Omron CX-Programmer project NewProject (CX-Programmer 9.76)

# PLC LQK19011ICM: CP1H XA
I/O table (CPU CP1H-XA40DR-A): rack 0 slot 0 CJ1W-SCU21

## Global symbols (name address type ; comment)
AI_SAW_CURRENT 200 CHANNEL  ; ANALOG.INPUT1.SAW.CURRENT
AI_TRANS_AXIS_DRIVE_VEL_FDBK 201 CHANNEL  ; AI.TRANSVERSE.AXIS.DRIVE.VELOCITY.FEEDBACK
AO_TRANS_VEL_REF 210 CHANNEL  ; TRANSVERSE.AXIS.VELOCITY.ANALOG.REFERENCE
0.05 BOOL  ; SPARE - Possible Zone Interference Limit Switch Input.
101 CHANNEL  ; @+ D205 &4 D205
1.03 BOOL  ; Spare
200 CHANNEL  ; Saw Motor Current Input
210 CHANNEL  ; Cross Travel Speed Refernce Command
40 CHANNEL  ; OI.SCALING.SAW.CURRENT.PART1
8.00 BOOL  ; Place holder for Automatic PID control request
A434.04 BOOL  ; Analog IO Initialised
D10009 CHANNEL  ; Spare
D1001 CHANNEL  ; Block 1 Data - Number of Blocks
D11040 CHANNEL  ; Operation Program Check Block 1 Slab 5 ID
D11050 CHANNEL  ; Operation Program Check Slab 6 ID
D11060 CHANNEL  ; Operation Program Check Slab ID
D11070 CHANNEL  ; Operation Program Check Slab 8 ID
D11080 CHANNEL  ; Operation Program Check Slab 9 ID
D11090 CHANNEL  ; Operation Program Check Slab 10 ID
D11100 CHANNEL  ; Operation Block 3 Slab 1 ID
D11110 CHANNEL  ; Operation Program Check Block 3 Slab 2 ID
D11120 CHANNEL  ; Operation Block 3 Slab 3 ID
D12301 CHANNEL  ; Operation Slab 31 Quantity
D12302 CHANNEL  ; Operation Program Check Block 7 Slab 31 Width
D200 CHANNEL  ; Number of Blocks Stored
D2002 CHANNEL  ; OPERATION.PROGRAM.CHECK.BLOCK1.SLAB2.SIZE
D201 CHANNEL  ; Operation Number of Words to Xfer
D202 CHANNEL  ; Captured Bumber of Blocks
D203 CHANNEL  ; Number of Blocks Difference
D204 CHANNEL  ; Slab Count Offset
D205 CHANNEL  ; Slab Word Count to Transfer
D3000 CHANNEL  ; Input Data Table Control Word
D3001 CHANNEL  ; Maximum Anaolg Input Value (Xm)
D3002 CHANNEL  ; Y0
D3003 CHANNEL  ; X1
D3004 CHANNEL  ; Maximum Output value
D3100 CHANNEL  ; Output Data Control Word
D3101 CHANNEL  ; Xm
D3102 CHANNEL  ; Y0
D3103 CHANNEL  ; X1
D3104 CHANNEL  ; Y1
D3106 CHANNEL  ; Interin feed rate calc word
D32 CHANNEL  ; OPERATION.AUTO.CYCLE.BLOCK.FIRST.CUT.WORKING.REAL
D3200 CHANNEL  ; Setpoint Input Data Table Control Word
D3201 CHANNEL  ; Maximum Input Setpoint
D3202 CHANNEL  ; Y0
D3203 CHANNEL  ; X1
D3204 CHANNEL  ; Y1
D34 CHANNEL  ; OP.CONTROL.VERTICAL.TARGET.SCALED
D3520 CHANNEL  ; PID Setpoint Scaled for PID
D3521 CHANNEL  ; PID Instruction Proportional Component
D3522 CHANNEL  ; PID Instruction Integral Component
D3523 CHANNEL  ; PID Instruction Derivative Component
D3524 CHANNEL  ; PID Instruction Period
D3525 CHANNEL  ; PID Instruction Control Word
D3526 CHANNEL  ; PID Instruction Input and Output Range Setting
D3527 CHANNEL  ; PID Instruction Output Minimum
D3528 CHANNEL  ; PID Instruction Output Maximum
D36 CHANNEL  ; OPERATION.AUTO.CYCLE.VERTICAL.HIGH/LOW/SPEED.SELECT
D40 CHANNEL  ; OP.CONTROL.CURRENT.BLOCK.HEIGHT.REAL
D400 CHANNEL  ; Working Floating Point First Cut Value Current Block
D4000 CHANNEL  ; OPERATION.AUTO.CYCLE.BLK.PTR
D4002 CHANNEL  ; OPERATION.AUTO.CYCLE.BLOCK.DATA.POINTER
D4004 CHANNEL  ; OPERATION.CURRENT.PROGRAM.SLAB.DATA.POINTER
D4006 CHANNEL  ; OPERATION.AUTO.CYCLE.SPARE
D4008 CHANNEL  ; OPERATION.AUTO.CYCLE.SPARE
D4010 CHANNEL  ; OPERATION.SLAB.POINTER.THIS.BLOCK
D4012 CHANNEL  ; OPERATION.AUTO.CYCLE.CURRENT.SLAB.CUT.COUNTER
D4014 CHANNEL  ; OPERATION.AUTO.CYCLE.SLAB.POINTER
D42 CHANNEL  ; OP.CONTROL.CURRENT.BLOCK.LENGTH
D44 CHANNEL  ; OP.CONTROL.AUTO.CYCLE.VERTICAL.TARGET
D46 CHANNEL  ; OP.CONTROL.AUTO.TRANSVERSE.TARGET.FORWARD
D48 CHANNEL  ; OP.CONTROL.TRANSVERSE.POSITION.TARGET.REAL
D480 CHANNEL  ; Ctl.PID.Output.Value
D484 CHANNEL  ; Saw Current Scaled for PID instruction use
D50 CHANNEL  ; OPERATION.AUTO.CYCLE.BLOCK.HEIGHT.REAL
D500 CHANNEL  ; First Cut Position Stored Float
D502 CHANNEL  ; Stored Slab Size Inches Float
D504 CHANNEL  ; Total Slab Size Float
D506 CHANNEL  ; Stored Kerf Size Total
D508 CHANNEL  ; Slab Total Size Calc'd
D510 CHANNEL  ; Total of First Cut Position and Slab Size
D512 CHANNEL  ; Final Calculated Position at Cut Finish of this Slab and this Block
D5120 CHANNEL  ; OI Long Axis Target
D52 CHANNEL  ; OPERATION.AUTO.CYCLE.BLOCK.TRANSVERSE.AXIS.FORWARD.STOP.POSITION
D5200 CHANNEL  ; Operation Long Axis Target Minimum
D54 CHANNEL  ; OPERATION.AUTO.CYCLE.BLOCK.FIRST.CUT.REAL
D5400 CHANNEL  ; OPERATION.LONG.TRAVEL.TARGET.WINDOW.PLUS
D5402 CHANNEL  ; OPERATION.LONG.TRAVEL.TARGET.WINDOW.MINUS
D5404 CHANNEL  ; OPERATION.LONG.TRAVEL.TARGET.WINDOW.SLABCUT.PLUS
D5406 CHANNEL  ; OPERATION.LONG.TRAVEL.TARGET.SLABCUT.MINUS
D5500 CHANNEL  ; OPERATION.AUTO.CYCLE.BLOCK.FIRST.CUT.REAL.SCALED
D5502 CHANNEL  ; OPERATION.AUTO.CYCLE.LON.INDEX.LOCATION.REAL.SCALED
D56 CHANNEL  ; OPERATION.AUTO.CYCLE.LONG.TARGET.KERF
D5600 CHANNEL  ; MC.TRANSVERSE.AXIS.POSITION.FEEDBACK.GB.SCALED.REAL
D58 CHANNEL  ; OPERATION.AUTO.CYCLE.ADD.KERF.TO.LOCATION.REAL
D6 CHANNEL  ; OPERATION.TRANSVERSE.AXIS.JOG.VELOCITY.REFERNCE.WORD
D60 CHANNEL  ; OPERATION.AUTO.CYCLE.LONG.INDEX.LOCATION.REAL
D6000 CHANNEL  ; MC.TRANSVERSE.AXIS.POSITION.FEEDBACK.RAW.REAL
D6002 CHANNEL  ; MC.TRANSVERSE.AXIS.POSITION.FEEDBACK.GB.SCALED.REAL
D6004 CHANNEL  ; MC.TRANSVERSE.AXIS.POSITION.PINION.REVOLUTIONS.REAL
D6006 CHANNEL  ; PI.EQUATION.PART.ONE
D6008 CHANNEL  ; PI.EQUATION.PART.TWO
D6012 CHANNEL  ; PI
D6014 CHANNEL  ; MC.TRANSVERSE.AXIS.PINION.CIRCUMFERENCE.INCHES.REAL
D66 CHANNEL  ; OPERATION.AUTO.CYCLE.CURRENT.SLAB.SIZE.REAL.RAW
D76 CHANNEL  ; OP.TRANSVERSE.AXIS.FORWARD.TARGET
D80 CHANNEL  ; Blade Kerf Raw Converted
D82 CHANNEL  ; Cut Depth Raw Converted
D84 CHANNEL  ; Cut Target Current Raw Converted
D86 CHANNEL  ; Current Slab Size Raw Converted
D97 CHANNEL  ; OP.CONTROL.AUTO.CYCLE.CURRENT.FIRST.CUT.LOCATION.LONG
D990 CHANNEL  ; PID Setpoint
H0.05 BOOL  ; OPERATION.ALARM.STATE.VALID
H0.11 BOOL  ; OPERATION.ALARM.RESET.COMMAND
H10.13 BOOL  ; MC.LONG.AXIS.STATE.VALID
H11.03 BOOL  ; VERTICAL.AXIS.DRIVE.NOT.OKAY
H11.07 BOOL  ; MC.VERTICAL.AXIS.JOG.PLUS
H11.08 BOOL  ; MC.VERTICAL.AXIS.JOG.MINUS
H11.13 BOOL  ; MC.VERTICAL.AXIS.DRIVE.RESET.ENABLED
H12.07 BOOL  ; MC.TRANSVERSE.AXIS.JOG.PLUS.INT
H12.08 BOOL  ; MC.TRANSVERSE.AXIS.JOG.NEG
H12.13 BOOL  ; MC.TRANSVERSE.AXIS.DRIVE.RESET.ENABLED
H13.04 BOOL  ; SAW.AUTO.RUN.UP.TIMER.DONE
H13.05 BOOL  ; OPERATION.AUTO.CYCLE.SAW.OVERCURRENT.ALARM
H13.06 BOOL  ; OPERATION.SAW.CURRENT.SENSING.CHECK.FAULT
H13.07 BOOL  ; OPERATION.SAW.MACHINE.STOP.COMMAND.ACTIVE
H13.08 BOOL  ; OPERATION.SAW.MACHINE.STOP.COMMAND.NOT ACTIVE
H13.13 BOOL  ; OPERATION.SAW.STATE.VALID
H13.15 BOOL  ; OP.ALARM.SAW.SOFT.START.FAULTED
H14.02 BOOL  ; WATER.FLOW.SHOULD.BE.ON
H14.03 BOOL  ; WATER.FLOW.IS.ON.AND.SHOULDN'T
H14.07 BOOL  ; OP.WATER.MACHINE.STOP.COMMAND.ACTIVE
H14.08 BOOL  ; OP.WATER.MACHINE.sTOP.COMMAND.NOT.ACTIVE
H14.13 BOOL  ; OPERATION.WATER.STATE.VALID
H14.14 BOOL  ; OP.ALARM.WATER.FLOW.ERROR
H16.13 BOOL  ; OPERATION.RECIPE.STATE.VALID
H16.14 BOOL  ; RECIPE.ERROR
H17.00 BOOL  ; Operation Auto Cycle State Invalid Over Time Alarm
H1.00 BOOL  ; OP.MODE.INDICATOR.ENABLED
H1.01 BOOL  ; OP.MODE.AUTO.PGM.CHECK.ACT
H1.02 BOOL  ; OP.MODE.AUTO.PGM.CHECK.CMP
H1.03 BOOL  ; LAST.BLOCK.CHECK
H1.14 BOOL  ; ALARM.RESEST.TRAP
H1.15 BOOL  ; MODE.AUTO.GATE.ALARM.TRIGGER
H2 CHANNEL  ; Cycle Start Bits
H20.04 BOOL  ; OPERATION.AUTO.CYCLE.LONG.AXIS.MOTION.READY
H20.05 BOOL  ; OPERATION.AUTO.CYCLE.LONG.AXIS.MOTION.ENABLED
H20.06 BOOL  ; OP.CONTROL.AUTO.CYCLE.INDEX.LONG.AXIS.COMMAND
H20.07 BOOL  ; OPERATION.AUTO.CYCLE.LONG.AXIS.INDEX.COMMAND.ACTIVE
H20.08 BOOL  ; OPERATION.LONG.AXIS.IN.POSITION.WINDOW.TOLERANCE
H20.09 BOOL  ; OPERATION.AUTO.CYCLE.LONG.AXIS.INDEX.COMMAND.COMPLETE
H20.10 BOOL  ; OPERATION.AUTO.CYCLE.LONG.AXIS.MOTION.SAFE
H20.11 BOOL  ; OPERATION.AUTO.CYCLE.LONG.AXIS.MOTION.COMMAND.RESET
H20.12 BOOL  ; OP.LONG.AXIS.MACHINE.STOP.ACTIVE
H20.13 BOOL  ; OPERATION.LONG.AXIS.MACHINE.STOP.NOT.ACTIVE
H20.14 BOOL  ; OP.CONTROL.INTERLOCK.LONG.AXIS.IN.MOTION
H20.15 BOOL  ; OPERATION.LONG.AXIS.MOTION.COMMAND.ERROR
H21.04 BOOL  ; Motion - Vertical Axis Motion Monitor enabled
H21.05 BOOL  ; MC.VERTICAL.AXIS.HOME.INIT
H21.06 BOOL  ; Motion - Vertical Axis Following Error Exists
H21.07 BOOL  ; MC_Vertical Axis Motion Error
H21.08 BOOL  ; OP.CONTROL.VERTICAL.IN.POSITION
H21.09 BOOL  ; OP.CONTROL.VERTICAL.HIGH.SPEED.SELECT
H21.10 BOOL  ; OP.CONTROL.VERTICAL.TARGET.CALC
H21.12 BOOL  ; OP.VERTICAL.AAXIS.MACHINE.STOP.ACTIVE
H21.13 BOOL  ; OP.VERTICAL.AXIS.MACHINE.STOP.NOT.ACTIVE
H21.14 BOOL  ; OP.CONTROL.INTERLOCK.VERTICAL.AXIS.IN.MOTION
H21.15 BOOL  ; MC.VERTICAL.AXIS.STATE.VALID
H22.05 BOOL  ; MC.TRANSVERSE.AXIS.HOMING.REQUEST
H22.06 BOOL  ; OPERATION.AUTO.TRANSVERSE.AXIS.IN.FORWARD.POSITION
H22.07 BOOL  ; Transverse Axis Following Error Fault
H22.08 BOOL  ; OP.CONTROL.AUTO.CYCLE.TRANSVERSE.AXIS.MOTION.ENABLE
H22.09 BOOL  ; Transverse Axis Following Error
H22.10 BOOL  ; OP.CONTROL.TRANSVERSE.TARGET.CALC
H22.12 BOOL  ; OP.TRANSVERSE.AXIS.MACHINE.STOP.ACTIVE
H22.13 BOOL  ; OP.TRANSVERSE.AXIS.MACHINE.STOP.NOT.ACTIVE
H22.14 BOOL  ; OP.CONTROL.INTERLOCK.TRANS.AXIS.IN.MOTION
H22.15 BOOL  ; MC.TRANSVERSE.AXIS.STATE.VALID
H2.00 BOOL  ; CYCLE.START.ENABLE
H2.01 BOOL  ; CYCLE.START.FUNCTION.RESET
H2.02 BOOL  ; CYCLE.START.FUNCTION.ENABLED
H2.03 BOOL  ; CYCLE.START.ACTIVE
H2.04 BOOL  ; CYCLE.START.COMPLETE
H2.05 BOOL  ; OPERATION.AUTO.CYCLE.START.COMMAND
H2.13 BOOL  ; OPERATION.CYCLE.START.STATE.VALID
H2.14 BOOL  ; CYCLE.START.ERROR
H32.07 BOOL  ; OPERATION.PROGRAM.CHECK.BLOCK1.ENABLE
H32.08 BOOL  ; OPERATION.PROGRAM.CHECK.BLOCK1.ENABLE
H32.09 BOOL  ; OPERATION.PROGRAM.CHECK.BLOCK2.ENABLE
H32.10 BOOL  ; OPERATION.PROGRAM.CHECK.BLOCK3.ENABLE
H32.11 BOOL  ; Operation Program Check Block 4 Enable
H32.12 BOOL  ; Operation Program Check Block 5 Enable
H32.13 BOOL  ; Operation Program Check Block 6 Enable
H32.14 BOOL  ; Operation Program Check Block 7 Enable
H32.15 BOOL  ; Operation Program Check Block 8 Enable
H33.00 BOOL  ; Operation Block 9 Enable
H33.01 BOOL  ; Operation Block 10 Enable Display
H33.02 BOOL  ; Operation Program Check Block 11 Enable Display
H33.03 BOOL  ; Operation Program Check Block 12 Enable Display
H35.00 BOOL  ; OPERATION.PROGRAM.CHECK.BLOCK1.ENABLE
H3.00 BOOL  ; OP_CTL_CYCLE_RUN_ENABLE
H3.01 BOOL  ; OP.CONTROL.CYCLE.RUN.ENABLED
H3.02 BOOL  ; CYCLE.RUN.ACTIVE
H3.03 BOOL  ; MACHINE.CYCLE.STOP
H3.04 BOOL  ; CYCLE.STOP.COMMAND
H3.05 BOOL  ; OPERATION.AUTO.CYCLE.STOP.COMMAND
H3.06 BOOL  ; OPERATION.CYCLE.RUN.RESET
H3.07 BOOL  ; OP.AUTO.CYCLE.ALARM.STATE.TRAP
H3.10 BOOL  ; OPERATION.AUTO.CYCLE.SEQUENCE.STEP.TIMER.DONE
H3.12 BOOL  ; OPERATION.MACHINE.STOP.STATE.VALID
H3.13 BOOL  ; OPERATION.AUTO.RUN.STATE.VALID
H3.14 BOOL  ; CYCLE.RUN.ERROR
H3.15 BOOL  ; Cycle Completed
H4 CHANNEL  ; Cycle Stop Bits
H4.00 BOOL  ; CYCLE.STOP.ENABLE
H4.01 BOOL  ; CYCLE.STOP.INSTRUCTION.RESET
H4.02 BOOL  ; CYCLE.STOP.FUNCTION.ENABLE
H4.03 BOOL  ; CYCLE.STOP.ACTIVE
H4.04 BOOL  ; CYCLE.STOP.COMPLETE
H4.05 BOOL  ; OPERATION.AUTO.CYCLE.ISSUE.SAFE.TO.STOP.COMMAND
H4.08 BOOL  ; OPERTION.CYCLE.STOP.COMMAND.INITIATED
H4.13 BOOL  ; OPERATION,CYCLE.STOP.STATE.VALID
H4.14 BOOL  ; CYCLE.STOP.INSTRUCTION.ERROR
H5.03 BOOL  ; GLOBAL.HOME.REQUEST.ACTIVE
H5.13 BOOL  ; Operation Global Home Request Valid State
H5.14 BOOL  ; Operation Auto Cycle Block Data Transfer Valid
H5.15 BOOL  ; Operation Slab Data Transfer Valid
H7 CHANNEL  ; Auto Cycle Step Word 1
H70 CHANNEL  ; OP.AUTO.CYCLE.STEP.STATE.TRAP
H7.00 BOOL  ; OPERATION.AUTO.CYCLE.SEQUENCE.STEP1
H7.01 BOOL  ; OPERATION.AUTO.CYCLE.SEQUENCE.STEP2
H7.02 BOOL  ; OPERATION.AUTO.CYCLE.SEQUENCE.STEP3
H7.03 BOOL  ; OPERATION.AUTO.CYCLE.SEQUENCE.STEP4
H7.04 BOOL  ; OPERATION.AUTO.CYCLE.SEQUENCE.STEP5
H7.05 BOOL  ; OPERATION.AUTO.CYCLE.SEQUENCE.STEP6
H7.06 BOOL  ; OPERATION.AUTO.CYCLE.SEQUENCE.STEP7
H7.07 BOOL  ; OPERATION.AUTO.CYCLE.SEQUENCE.STEP8
H7.08 BOOL  ; OPERATION.AUTO.CYCLE.SEQUENCE.STEP9
H7.09 BOOL  ; OPERATION.AUTO.CYCLE.SEQUENCE.STEP10
H7.10 BOOL  ; OPERATION.AUTO.CYCLE.SEQUENCE.STEP11
H7.11 BOOL  ; OPERATION.AUTO.CYCLE.SEQUENCE.STEP12
H7.12 BOOL  ; OPERATION.AUTO.CYCLE.SEQUENCE.STEP13
H7.13 BOOL  ; OPERATION.AUTO.CYCLE.SEQUENCE.STEP14
H7.14 BOOL  ; OPERATION.AUTO.CYCLE.SEQUENCE.STEP15
H7.15 BOOL  ; OPERATION.AUTO.CYCLE.SEQUENCE.STEP16
H8 CHANNEL  ; Auto Cycle Step Word 2
H8.00 BOOL  ; OPERATION.AUTO.CYCLE.SEQUENCE.STEP17
H8.01 BOOL  ; OPERATION.AUTO.CYCLE.SEQUENCE.STEP18
H8.02 BOOL  ; OPERATION.AUTO.CYCLE.SEQUENCE.STEP19
H8.03 BOOL  ; OPERATION.AUTO.CYCLESEQUENCE.STEP20
H8.04 BOOL  ; OPERATION.AUTO.CYCLE.SEQUENCE.STEP21
H8.05 BOOL  ; OPERATION.AUTO.CYCLE.SEQUENCE.STEP22
H8.06 BOOL  ; OPERATION.AUTO.CYCLE.SEQUENCE.STEP23
H8.07 BOOL  ; OPERATION.AUTO.CYCLE.SEQUENCE.STEP24
H8.08 BOOL  ; OPERATION.AUTO.CYCLESEQUENCE.STEP25
H8.09 BOOL  ; OPERATION.AUTO.CYCLE.SEQUENCE.STEP26
H8.10 BOOL  ; OPERATION.AUTO.CYCLE.SEQUENCE.STEP27
H9 CHANNEL  ; OPERATION.AUTO.CYCLE.SEQUENCE.STATE.BITS
H9.00 BOOL  ; Operation First Cut is completed
H9.01 BOOL  ; Operation Block is Completed
H9.02 BOOL  ; OPERATION.AUTO.CYCLE.CURRENT.BLOCK.NO.SLABS.BIT
H9.03 BOOL  ; OPERATION.AUTO.CYCLE.ZERO.HEGHTBLOCK
H9.04 BOOL  ; Operation Zero Slab Width - Cycle Stop
H9.10 BOOL  ; OPERATION.AUTO.CYCLE.SEQUENCE.STEP.ENABLE
H9.11 BOOL  ; Operation Auto Cycle Step Allow
H9.12 BOOL  ; OPERATION.AUTO.CYCLE.SEQUENCE.STEP.ERROR
H9.13 BOOL  ; OPERATION.AUTO.CYCLE.SEQUENCE.STATE.ENABLED
H9.14 BOOL  ; OPERATION.SEQUENCE.STATE.INVALID
H9.15 BOOL  ; OPERATION.AUTO.CYCLE.SEQUENCE.STATE.VALID
T0000 BOOL  ; Step 0 Timer Done
T0001 BOOL  ; Step 1 Timer Done
T0002 BOOL  ; Step 2 timer done
T0003 BOOL  ; Increment Slab Pulse Timer
T0004 BOOL  ; Slab Decrement Pulse Timer
T0005 BOOL  ; Block Increment Pulse Timer
T0006 BOOL  ; Block Decrement Pulse Timer
T0010 BOOL  ; Block Step 0 Timer
T0011 BOOL  ; Block Step 1 Timer
T0012 BOOL  ; Block Step 2 Timer
T0013 BOOL  ; Block Step 3 Timer
T0014 BOOL  ; Block Step 4 timer
T0015 BOOL  ; Block Step 5 Timer
T0016 BOOL  ; Block Step 6 Timer
T0017 BOOL  ; Saw Current At Limit Timer
T0018 BOOL  ; OPERATION.SAW.CURRENT.SENSING.ZERO.CURRENT.CHECK.TIMER
T0019 BOOL  ; MC_Vertical Axis Motion Monitor Timer
T0020 BOOL  ; MC.VERTICAL.AXIS.BRAKE.TIMER
T0021 BOOL  ; MC.LONG.AXIS.HOME.ACT.TIMER
T0022 BOOL  ; MC.LONG.AXIS.INDEX.COMMAND.COMPLETE.TIME
T0023 BOOL  ; Index Position Data Setle Timer
T0024 BOOL  ; Transverse Axis Motion Error Timer
T0029 BOOL  ; OPERATION.AUTO.CYCLE.SEQUENCE.STEP1.TIMER
T0030 BOOL  ; OPERATION.AUTO.CYCLE.STEP2.TIMER
T0031 BOOL  ; OPERATION.SEQUENCE.STEP3.TIMER
T0032 BOOL  ; OPERATION.AUTO.CYCLE.SEQUENCE.STEP4.TIMER
T0033 BOOL  ; OPERATION.AUTO.CYCLE.SEQUENCE.STEP5.TIMER
T0034 BOOL  ; OPERATION.AUTO.CYCLE.SEQUENCE.STEP6.TIMER
T0035 BOOL  ; OPERATION.AUTO.CYCLE.SEQUENCE.STEP7.TIMER
T0036 BOOL  ; OPERATION.AUTO.CYCLE.SEQUENCE.STEP8.TIMER
T0037 BOOL  ; OPERATION.AUTO.CYCLE.SEQUENCE.STEP9.TIMER
T0038 BOOL  ; OPERATION.AUTO.CYCLE.SEQUENCE.STEP10.TIMER
T0039 BOOL  ; OPERATION.AUTO.CYCLE.SEQUENCE.STEP11.TIMER
T0040 BOOL  ; OPERATION.AUTO.CYCLE.SEQUENCE.STEP12.TIMER
T0041 BOOL  ; OPERATION.AUTO.CYCLE.SEQUENCE.STEP13.TIME
T0042 BOOL  ; OPERATION.AUTO.CYCLE.STEP14.TIMER
T0043 BOOL  ; OPERATION.AUTO.CYCLE.STEP15.TIMER
T0044 BOOL  ; OPERATION.AUTO.CYCLE.SEQUENCE.STEP16.TIMER
T0045 BOOL  ; OPERATION.AUTO.CYCLE.SEQUENCE.STEP17.TIMER
T0046 BOOL  ; OPERATION.AUTO.CYCLE.SEQUENCE.STEP18.TIMER
T0047 BOOL  ; OPERATION.AUTO.CYCLE.SEQUENCE.STEP19.TIMER
T0048 BOOL  ; OPERATION.AUTO.CYCLE.SEQUENCE.STEP20.TIMER
T0049 BOOL  ; OPERATION.AUTO.CYCLE.SEQUENCE.STEP21.TIMER
T0050 BOOL  ; OPERATION.AUTO.CYCLE.SEQUENCE.STEP22.TIMER
T0051 BOOL  ; OPERATION.AUTO.CYCLE.SEQUENCE.STEP23.TIMER
T0052 BOOL  ; OPERATION.AUTO.CYCLE.STEP24.TIMER
T0053 BOOL  ; OPERATION.AUTO.CYCLE.SEQUENCE.STEP25.TIMER
T0054 BOOL  ; OPERATION.AUTO.CYCLE.SEQUENCE.STEP26.TIMER
T0055 BOOL  ; OPERATION.AUTO.CYCLE.SEQUENCE.STEP27.TIMER
T0090 BOOL  ; Operation Auto Cycle Sequence Step Error Timer
T0100 BOOL  ; Index Delay Time
T0101 BOOL  ; OPERATION.LONG.AXIS.INDEX.COMMAND.START.DELAY.TIMER
T0102 BOOL  ; OPERATION.AUTO.CYCLE.LONG.AXIS.FIRST.CUT.LOADED.TIMER
T0103 BOOL  ; OPERATION.AUTO.CYCLE.LONG.AXIS.INDEX.POSITION.LOADED.TIMER
T0130 BOOL  ; OPERATION.AUTO.CYCLE.SAW.RUN.UP.TIME
T0140 BOOL  ; WATER.FAULT.TIMER
T0200 BOOL  ; OPERATION.CONTROL.RESET.SEQUENCE.TIMER
W0.01 BOOL  ; Test Bit Blocker. Remove when done
W0.02 BOOL  ; OPERATION.AUTO.MODE.SELECTED.WITH.SAFETY.GATE.OPEN
W0.12 BOOL  ; GLOBAL.HOME.REQUEST.HOME.TRANSVERSE
W0.13 BOOL  ; GLOBAL.HOME.REQUEST.HOME.VERTICAL
W0.14 BOOL  ; CTL.GLOBAL.HOME.REQUEST.COMPLETED
W102.00 BOOL  ; OI.MESSAGE.INTERNAL.TRIGGER.MSG1
W102.01 BOOL  ; OI.MESSAGE.MSG2.TRIGGER
W102.02 BOOL  ; OI.MESSAGE.MSG3.TRIGGER
W102.03 BOOL  ; OI.MESSAGE.MSG4.TRIGGER
W102.04 BOOL  ; OI.MESSAGE.MSG5.TRIGGER
W102.05 BOOL  ; OI.MESSAGE.MSG6.TRIGGER
W102.06 BOOL  ; OI.MESSAGE.MSG7.TRIGGER
W102.07 BOOL  ; OI.MESSAGE.MSG8.TRIGGER
W102.08 BOOL  ; OI.MESSAGE.MSG9.TRIGGER
W102.09 BOOL  ; OI.MESSAGE.MSG10.TRIGGER
W104.00 BOOL  ; OI.MESSAGES.ENABLED
W104.01 BOOL  ; OI.MESSAGE.MSG2.ENABLED
W104.15 BOOL  ; OI.GLOBAL.MESSAGE.TRIGGER
W108 CHANNEL  ; OI.MESSAGE.COLOUR.INTERNAL
W109 CHANNEL  ; OI.MESSAGE.SELECT.INTERNAL
W110.00 BOOL  ; Alarm Message Trigger - Main Power Loss
W110.01 BOOL  ; Alarm Message Trigger - Safety Gate Open in Auto Mode
W110.02 BOOL  ; Alarm Message Trigger - Long Travel Axis Drive Error
W110.03 BOOL  ; Alarm Message Trigger - Vertical Axis Drive Error
W110.04 BOOL  ; Alarm Message - Transverse Axis Drive Error
W110.05 BOOL  ; Alarm Message Trigger - Saw Motor Current Sensor Error
W110.09 BOOL  ; Alarm Message Trigger - Program Check Error
W110.12 BOOL  ; Alarm Message Trigger - Saw Soft Start Trip Error
W110.13 BOOL  ; Alarm Message Trigger - Saw Over Current/Blade Pinch Error
W111.05 BOOL  ; Alarm Message Trigger - Water Should be On Error
W111.06 BOOL  ; Alarm Message Trigger - Water Should be Off Error
W111.15 BOOL  ; Alarm Message Trigger - Transverse Drive Mains Loss
W112.00 BOOL  ; Alarm Message Trigger - Transverse Drive Overload Error
W112.01 BOOL  ; Alarm Message Trigger - Transverse Drive Over Temperature Error
W112.02 BOOL  ; Alarm Messae Trigger - Transverse drvive general error
W112.03 BOOL  ; OI.ALARM.MESSAGE.MSG4.TRIGGER
W112.04 BOOL  ; OI.ALARM.MESSAGE.MSG5.TRIGGER
W112.05 BOOL  ; OI.ALARM.MESSAGE.MSG6.TRIGGER
W112.09 BOOL  ; OI.ALARM.MESSAGE.MSG10.TRIGGER
W112.10 BOOL  ; OI.ALARM.MESSAGE.MSG11.TRIGGER
W112.12 BOOL  ; OI.ALARM.MESSAGE.MSG13.TRIGGER
W112.13 BOOL  ; OI.ALARM.MESSAGE.MSG14.TRIGGER
W112.15 BOOL  ; OI.ALARM.MESSAGE.MSG16.TRIGGER
W113.05 BOOL  ; OI.ALARM.MESSAGE.MSG21.TRIGGER
W113.06 BOOL  ; OI.ALARM.MESSAGE.MSG22.TRIGGER
W113.07 BOOL  ; OI.ALARM.MESSAGE.MSG13.TRIGGER
W113.15 BOOL  ; OI.ALARM.MESSAGE.MSG31.TRIGGER
W114.00 BOOL  ; Alarm Message Trigger - Vertical Drive Mains Loss
W114.01 BOOL  ; Alarm Message Trigger - Vertical Drive Overload Error
W114.02 BOOL  ; Alarm Message Trigger - Vertical Drive Over Temperature Error
W114.03 BOOL  ; Alarm Messsage Trigger - Vertical Drive General Error
W114.04 BOOL  ; Vertical Axis Following Error
W114.15 BOOL  ; OI.ALARM.MESSAGE.TRIGGER.GLOBAL
W115 CHANNEL  ; OI.INTERNAL.ALARM.MESSAGE.SELECTION
W115.00 BOOL  ; Alarm Message Trigeer - Long Drive Mains Loss Error
W115.01 BOOL  ; Alarm Message Trigger - Long Drive Bus Under Voltage Error
W115.02 BOOL  ; Alarm Message Trigger - Long Drive Overload Error
W115.03 BOOL  ; Alarm Message Trigger - Long Drive Over Temperature Error
W115.04 BOOL  ; Alarm Message Trigger - Unspecified Alarm Exists on Long Drive
W115.05 BOOL  ; Alarm Message Triger - Auto Cycle Sequence Step Invalid State Over Time Alarm
W115.06 BOOL  ; Alarm Message Trigger - Zero Height Block Encountered, cycle stop initiated
W115.07 BOOL  ; Alarm Message Trigger - Zero width slab error, cycle stop initiated
W116.00 BOOL  ; OI.ALARM.MESSAGE.MSG51.TRIGGER
W116.01 BOOL  ; OI.ALARM.MESSAGE.MSG52.TRIGGER
W116.02 BOOL  ; OI.ALARM.MESSAGE.MSG53.TRIGGER
W116.03 BOOL  ; OI.ALARM.MESSAGE.MSG54.TRIGGER
W117.00 BOOL  ; OI.ALARM.MESSAGE.MSG71.TRIGGER
W117.01 BOOL  ; OI.ALARM.MESSAGE.MSG72.TRIGGER
W117.02 BOOL  ; OI.ALARM.MESSAGE.MSG73.TRIGGER
W117.03 BOOL  ; ALARM.MESSAGE.MSG74.TRIGGER
W117.04 BOOL  ; OI.ALARM.MESSAGE.MSG75.TRIGGER
W118 CHANNEL  ; OI.ALARM.MESSAGE.COLOUR.SELECT.INTERNAL
W120.09 BOOL  ; OI.VERTICAL.AXIS.HOME.REQUEST.PB
W121.02 BOOL  ; Previous Block
W121.03 BOOL  ; Previous Slab of Current Block
W121.04 BOOL  ; Next Slab of current Block
W121.05 BOOL  ; Next Block Select
W121.07 BOOL  ; Clear Data
W121.09 BOOL  ; OI.ALARM.ACCEPT.CONFIRMATION
W121.10 BOOL  ; OI.CONTROL.RESET.AUTO.CYCLE.SEQUENCE
W121.11 BOOL  ; OI.COONTROL.CONTINUE.AT.CURRENT.SEQUENCE.STEP.PB
W121.12 BOOL  ; OI.CONTROL.SKIP.CUT.AT.CURRENT.SEQUENCE.STEP
W121.13 BOOL  ; OI.CONTROL.SKIP.BLOCK.AT.CURRENT.SEQUENC.STEP
W12.00 BOOL  ; Slab Change Data Storage and Display Update Step 0
W12.01 BOOL  ; Step 1
W12.02 BOOL  ; Step 2
W12.03 BOOL  ; Step 3
W12.04 BOOL  ; Step 4
W12.05 BOOL  ; Step 5
W12.06 BOOL  ; Step 6
W12.15 BOOL  ; Loop Step Reset
W130.00 BOOL  ; OI.ALL.HOME.INDICATOR
W130.04 BOOL  ; OI.VERTICAL.AXIS.HOME.INDICATOR
W130.05 BOOL  ; OI.VERTICAL.AXIS.JOG.FORWARD.INDICATOR
W130.06 BOOL  ; OI.VERTICAL.AXIS.JOG.REVERSE.INDICATOR
W130.07 BOOL  ; OI.INDICATE.TRANSVERSE.AXIS.HOME.INDICATOR
W130.08 BOOL  ; OI.TRANSVERSE.AXIS.JOG.REVERSE.INDICATOR
W130.09 BOOL  ; OI.TRANSVERSE.AXIS.JOG.FORWARD.INDICATOR
W130.10 BOOL  ; OI.LONG.AXIS.JOG.RIGHT.COMMAND.ACTIVE.INDICATOR
W130.11 BOOL  ; OI.LONG.AXIS.JOG.LEFT.COMMAND.ACTIVE.INDICATOR
W130.12 BOOL  ; OI.LONG.AXIS.HOME.INDICATOR
W131.00 BOOL  ; OI.SLAB.INCREMENT.PB.ENABLE
W131.01 BOOL  ; OI.BLOCK.POINTER.INCREMENT.PB.ENABLE
W131.02 BOOL  ; OP.AUTO.CYCLE.ALARM.CONDITION.IN.CYCLE.MESSAGE.SHOW
W13.00 BOOL  ; Step 0 in Progress
W13.01 BOOL  ; Step 1 in Progress
W13.02 BOOL  ; Step 2 in Progress
W13.03 BOOL  ; Step 3 in Progress
W13.04 BOOL  ; Step 4 in Progress
W13.05 BOOL  ; Step 5 in Progress
W13.06 BOOL  ; Step 6 in Progress
W14.00 BOOL  ; Step 0 Done
W14.01 BOOL  ; Step 1 Done
W14.02 BOOL  ; Step 2 Done
W14.03 BOOL  ; Step 3 Done
W14.04 BOOL  ; Step 4 Done
W14.05 BOOL  ; Step 5 Done
W14.06 BOOL  ; Step 6 Done
W150 CHANNEL  ; Block Number Captured
W151 CHANNEL  ; Number of Words for Blocks
W152 CHANNEL  ; Slab Count Work Word for Block Pointer
W153 CHANNEL  ; Offset Calculate for Last Slab Count
W154 CHANNEL  ; Offset Mid Calc
W156 CHANNEL  ; Offset Calc'd
W158 CHANNEL  ; Slab Record Offset Interim
W15.00 BOOL  ; Block Change Data Storage and Display Update Step 0
W15.01 BOOL  ; Loop Step 1
W15.02 BOOL  ; Loop Step 2
W15.03 BOOL  ; Loop Step 3
W15.04 BOOL  ; Loop Step 4
W15.05 BOOL  ; Loop Step 5
W15.06 BOOL  ; Loop Step 6
W15.15 BOOL  ; Loop Step Reset
W160 CHANNEL  ; Slab Offset Result
W16.00 BOOL  ; Step 0 in Progress
W16.01 BOOL  ; Loop Step 1 in Progress
W16.02 BOOL  ; Loop Step 2 in Progress
W16.03 BOOL  ; Loop Step 3 in Progress
W16.04 BOOL  ; Loop Step 4 in Progress
W16.05 BOOL  ; Loop Step 5 in Progress
W16.06 BOOL  ; Loop Step 6 in Progress
W16.10 BOOL  ; Slab Data Read in Progress
W16.11 BOOL  ; Block Data Read in Progress
W17.00 BOOL  ; Step 0 Done
W17.01 BOOL  ; Loop Step 1 Done
W17.02 BOOL  ; Loop Step 2 Complete
W17.03 BOOL  ; Loop Sstep 3 Complete
W17.04 BOOL  ; Loop Step 4 Complete
W17.05 BOOL  ; Loop Step 5 Complete
W17.06 BOOL  ; Loop Step 6 Complete
W190 CHANNEL  ; Slab Pointer Offset Adjustment
W191 CHANNEL  ; Block 1 Slab Count Capture
W192 CHANNEL  ; Slab Offset Addition for This Block
W193 CHANNEL  ; Slab_ID_Raw
W194 CHANNEL  ; Slab Pointer Calculated
W195 CHANNEL  ; Slab Offset Previous
W196 CHANNEL  ; Slab_Offset_Constant_Calculated
W197 CHANNEL  ; Block_Selected_Base
W198 CHANNEL  ; Block Pointer Offset Calculated
W19.00 BOOL  ; Test Bit
W19.01 BOOL  ; Self Toggle
W1.01 BOOL  ; Test Bit 2
W1.02 BOOL  ; Operation Main Power Loss Error
W200 CHANNEL  ; Current Programming Block ID
W201 CHANNEL  ; Current Programming Number of Blocks
W205 CHANNEL  ; Current Programming Block First Cut Location
W209 CHANNEL  ; Spare
W20.00 BOOL  ; Block Incremented Pulse - Lead
W20.01 BOOL  ; Block Decremented Pulse - Lead
W20.02 BOOL  ; Slab Incremented Pulse - Lead
W20.03 BOOL  ; Slab Decremented Pulse - Lead
W20.04 BOOL  ; Slab Count Capture Trap
W20.05 BOOL  ; Block Read In Progress
W20.06 BOOL  ; Slab Count Changed from Block Read
W20.07 BOOL  ; Slab Pointer Updating
W20.08 BOOL  ; Update Working Offset
W20.09 BOOL  ; Block Pointer Calculate Enable
W20.10 BOOL  ; Increment Block Pointer
W20.11 BOOL  ; Decrement Block Pointer
W20.12 BOOL  ; First_Pass_Read
W20.14 BOOL  ; Block Offset Calculated
W20.15 BOOL  ; Block Program Control Enabled
W21.00 BOOL  ; Blade Kerf Data Write to Storage
W21.01 BOOL  ; Blade Kerf Read from Storage
W21.02 BOOL  ; Cut Depth Write to Storage
W21.03 BOOL  ; Cut Depth Read from Storage
W21.04 BOOL  ; Target Saw Current in Amps Write to Storage
W21.05 BOOL  ; Target Saw Current in Amps Read from Storage
W21.06 BOOL  ; Read Slab Data from Storage
W21.07 BOOL  ; Block Data Write to Storage
W21.08 BOOL  ; Automatic Number of Blocks Update
W21.09 BOOL  ; Slab Pointer Control Enabled
W21.10 BOOL  ; Increment Slab Offset
W21.11 BOOL  ; Decrement Slab Offset
W21.12 BOOL  ; Automatic Number of Slabs Update
W21.13 BOOL  ; Slab Pointer Reset
W21.14 BOOL  ; Block Pointer Reset
W22.00 BOOL  ; Slab Pointer Calculated
W22.01 BOOL  ; Block Pointer Changed
W22.02 BOOL  ; Current Block Selected Changed Initiate Block Data Write
W22.03 BOOL  ; Block Data Write Step Zero Complete
W22.04 BOOL  ; Block Data Write Complete
W22.05 BOOL  ; Capture Current Slab Words
W22.06 BOOL  ; Slab Data Write In Progress
W22.07 BOOL  ; Slab Data Write Complete
W22.08 BOOL  ; Block Offset Adjusted
W22.09 BOOL  ; Block Offset Adjust Complete
W22.10 BOOL  ; Block Data Read in Progress
W22.11 BOOL  ; Block Data Read >
W22.12 BOOL  ; Block Data Read Complete
W22.13 BOOL  ; Slab Offset Adjust in Progress
W22.14 BOOL  ; Slab Offset Adjust >
W22.15 BOOL  ; Slab Offset Adjust Complete
W23.00 BOOL  ; Slab Offset Init
W23.01 BOOL  ; Slab Offset Pointer Updating
W23.02 BOOL  ; Slab Offset Updated
W23.03 BOOL  ; Slab Data Read in Progress
W23.04 BOOL  ; Slab Data Read >
W23.05 BOOL  ; Slab Data Read Complete
W23.15 BOOL  ; Slab Offset Init Complete
W24.01 BOOL  ; Offset Init Step 1 Complete
W24.02 BOOL  ; OffsetInit Step 2 Complete
W24.03 BOOL  ; Offset Init Step 3 Complete
W250 CHANNEL  ; Offset value for Second word in indirect addressed storage area for Block Start Edge
W251 CHANNEL  ; Offset Value for Third word in Storge area for block length
W252 CHANNEL  ; Offset value calculated for 4th word in Storage area for block First Cut
W253 CHANNEL  ; Offset value calculated for number of slabs for current block
W256 CHANNEL  ; Last Slab Count from First Block
W257 CHANNEL  ; Offset adjust
W25.01 BOOL  ; Offset Init Step 1 In Progress
W25.02 BOOL  ; Offset Init Step 2 In Progress
W25.03 BOOL  ; Offset Init Step 3 In Progress
W26.00 BOOL  ; Minus Slab Offset Init
W26.01 BOOL  ; Minus Offset Init Step 1
W26.02 BOOL  ; Minus Offset Init Step 2
W26.03 BOOL  ; Minus Offset Init Step 3
W26.15 BOOL  ; Minus Slab Offset Init Complete
W27.01 BOOL  ; Minus Offset Init Step 1 Complete
W27.02 BOOL  ; Minus Offset Init Step 2 Complete
W27.03 BOOL  ; Minus Offset Init Step 3 Complete
W28.01 BOOL  ; Minus Offset Init Step 1 In Progress
W28.02 BOOL  ; Minus Offset Init Step 2 In Progress
W28.03 BOOL  ; Minus Offset Init Step 3 In Progress
W2.00 BOOL  ; Program Check - Increment Slab Pointer
W2.01 BOOL  ; Program Check - Increment Block
W2.02 BOOL  ; Program Check - Completed
W2.05 BOOL  ; Reset Pointer after Program Check
W300 CHANNEL  ; Blade Kerf Working
W301 CHANNEL  ; Cut Depth Working
W302 CHANNEL  ; Target Current Working
W30.00 BOOL  ; OI.MESSAGE.INTERNAL.TRIGGER.MSG1
W30.01 BOOL  ; OI.MESSAGE.INTERNAL.TRIGGER.MSG2
W30.09 BOOL  ; OI.ALARM.MESSAGE.TRIGGER.MSG10
W312 CHANNEL  ; Last Block ID
W313 CHANNEL  ; Current Block ID Stored
W314 CHANNEL  ; Last Programmed numer of blocks
W315 CHANNEL  ; Current Stored Number of Blocks
W31.00 BOOL  ; OI.MESSAGE.CONTROL.ENABLED
W320 CHANNEL  ; Current Block Last Number of Slabs
W321 CHANNEL  ; Current Block Stored Slab Count
W322 CHANNEL  ; Current Slab Last Width
W323 CHANNEL  ; Current Slab Stored Width
W324 CHANNEL  ; Current Slab Last Quantity
W325 CHANNEL  ; Current Slab Stored Quantity
W350 CHANNEL  ; Axis position display
W37.00 BOOL  ; Current and Previous Block ID are Different
W37.01 BOOL  ; Last Stored Block ID and Current Block ID are Different
W37.02 BOOL  ; Current Block Number of Blocks and Stored Number of Blocks are Not Equal
W37.03 BOOL  ; Last Block Number of Blocks and Stored Value are not equal
W37.04 BOOL  ; Current Block Height and Stored Block Height are different
W37.05 BOOL  ; Last Block Last and Stored Heights are different
W37.06 BOOL  ; Current and Stored Cross Stop not Equal
W37.07 BOOL  ; Last and Stored Cross Stop are not equal
W37.08 BOOL  ; Programmed and Stored Block First Cut not equal
W37.09 BOOL  ; Last and Stored Block First cur not equal
W37.10 BOOL  ; Block Current and Last Slab count are different
W37.11 BOOL  ; Current and Last Slab ID's are Not Equal
W37.12 BOOL  ; Last and Stored Slab ID are Not Equal
W37.13 BOOL  ; Current and Last Slab Cut Qty are Not Equal
W37.14 BOOL  ; Crrent and Stored Slab sizes are different
W37.15 BOOL  ; Last and Stored Slab Sizes are different
W38.00 BOOL  ; Current and Stored Slab Cut Quantity are not equal
W3.00 BOOL  ; STEP.ONE.EXECUTE
W3.01 BOOL  ; STEP.TWO.EXECUTE
W3.02 BOOL  ; STEP.THREE.EXECUTE
W400 CHANNEL  ; Temporary Storage for Block Data Used in Slab Offset Calc
W400.00 BOOL  ; Data Write Step
W400.01 BOOL  ; Data Offset Adjust Step
W400.02 BOOL  ; Data Read Step
W400.03 BOOL  ; End Step
W404 CHANNEL  ; # of Slabs for current Block
W405 CHANNEL  ; Number of words used by slabs in this block
W406 CHANNEL  ; Temporary Offset Storage word
W40.00 BOOL  ; Data Write/Read Sequence Initiate
W40.01 BOOL  ; Data Write Step Action
W40.02 BOOL  ; Data Offset Adjust Action
W40.03 BOOL  ; Data Read Step Action
W41.00 BOOL  ; Slab Data Write in Progress
W41.01 BOOL  ; Slab Data Write >
W41.02 BOOL  ; Slab Offset Adjust in Progress
W41.03 BOOL  ; Calulating Number of Words to Read
W4.00 BOOL  ; Program Check - Block First Cut Error
W4.01 BOOL  ; Program Check Step 1 - Block Pointer Reset
W4.02 BOOL  ; Program Check Step 1 - Ready for Next Step
W4.03 BOOL  ; Program Check Step 1 _ Store First Cut Position as Floating Point
W4.04 BOOL  ; Program Check Step 2 - Calculation Settle
W4.05 BOOL  ; Program Check Step 3 - Slab Size Convert to Floating Point
W4.06 BOOL  ; Program Check Step 3 - Totalise Kerf and Slab sizes Claculate Slab Size
W4.07 BOOL  ; Slab Size Calc
W4.08 BOOL  ; Calculate Kerf Total
W4.09 BOOL  ; Program Check Step 3 - Kerf Total Calculation
W4.10 BOOL  ; Program Check Step 3 - Add Kerf Total to Slab Size Total
W4.11 BOOL  ; Program Check Step 3 - Total Size Calculation => Position Target
W4.12 BOOL  ; Program Check Step 3 - Slab Inrement
W4.13 BOOL  ; Program Check Step 3 - Phase 2
W4.15 BOOL  ; Program Check Step 3 - Ready for Next Step
W5.00 BOOL  ; GLOBAL.HOME.REQUEST.HOME.LONG.TRAVEL
W5.01 BOOL  ; OPERATION.AUTO.CYCLE.SLAB.POINTER.INCREMENTED
W6.04 BOOL  ; OP.CONTROL.AUTO.CYCLE.RUN.EXECUTE.STEP2
W6.05 BOOL  ; OP.CONTROL.AUTO.CYCLE.RUN.STEP2
W6.06 BOOL  ; OP.CONTROL.AUTO.CYCLE.STEP3.RUN
W6.07 BOOL  ; OP.CONTROL.AUTO.CYCLE.RUN.STEP3.RAISE.VERTICAL
W6.08 BOOL  ; OP.CONTROL.RAISE.VERTICAL
W6.09 BOOL  ; OP.CONTROL.AUTO.CYCLE.STEP4
W6.10 BOOL  ; OP.CONTROL.AUTO.CYCLE.RUN.STEP4.INDEX.LONG
W7.00 BOOL  ; AUTO.MODE.ENABLED.RESET.WORKING.TO.FIRST.BLOCK
W7.03 BOOL  ; AUTO.SEQUENCE.STEP4.DN
W7.04 BOOL  ; Ctl.PID.Executing
W7.05 BOOL  ; Ctl.PID.Error
W7.06 BOOL  ; Current Position is Desired Position
W7.07 BOOL  ; MC.LONG.AXIS.INDEX.COMMAND.ACTIVE
W7.08 BOOL  ; MC.LONG.AXIS.INDEX.COMMAND.COMPLETED
W7.09 BOOL  ; OP.CONTROL.AUTO.CYCLE.RUN.SAW.MOTION
W7.10 BOOL  ; OP.CONTROL.INDEX.LONG
W8.00 BOOL  ; Place holder for auto index action Testing
W8.01 BOOL  ; OPERATION.STEP1.BLOCK.DATA.READ.ACTIVE
W8.02 BOOL  ; OPERATION.AUTO.CYCLE.SLAB.DATA.READ.ACTIVE
W8.03 BOOL  ; Place Holder for Incrementing (if required) Block Pointer
W8.04 BOOL  ; OPERATION.AUTO.CYCLE.SLAB.POINTER.ENABLED
W8.05 BOOL  ; OPERATION.STEP2.CALCULATE.POSITIONS
W8.06 BOOL  ; OPERATION.AUTO.CYCLE.STEP2.CALCULATE.CROSS.FORWARD.POSITION
W8.07 BOOL  ; OPERATION.AUTO.CYCLE.STEP2.CALCULATE.FIRST.CUT.POSITION
W8.08 BOOL  ; OPERATION.AUTO.CYCLE.STEP7.CALACULATE.SLAB.SIZE
W8.09 BOOL  ; OPERATION.MOVE.BLOCK.HEIGHT.TO.VERTICAL.TARGET
W8.10 BOOL  ; OPERATION.AUTO.CYCLE.SEQ.STEP5.CALULATE.CUT.HEIGHT
W8.11 BOOL  ; OPERATION.AUTO.CYCLE.CALCULATE.LONG.TARGET.PART1
W8.12 BOOL  ; OPERATION.AUTO.CYCLE.CALCULATE.FINAL.LONG.TARGET
W8.13 BOOL  ; OPERATION.AUTO.CYCLE.LAST.CUT.FOR.CURRENT.SLAB
W8.14 BOOL  ; OPERATION.AUTO.CYCLE.CURRENT.SLAB.COUNTED.EQUALS.SLAB.QTY
W8.15 BOOL  ; OPERATION.AUTO.CYCLE.INC.SLAB.PTR
W90.00 BOOL  ; Block Data Write Step 0
W90.01 BOOL  ; Slab Data Write Step 1
W90.02 BOOL  ; Change Block Offset Pointer
W90.03 BOOL  ; Read Block Data
W90.04 BOOL  ; Slab Offset Adjust
W90.05 BOOL  ; Slab Offset Pointer Update
W90.06 BOOL  ; Slab Data Read
W90.07 BOOL  ; Last Step
W9.00 BOOL  ; OPERATION.AUTO.CYCLE.DEC.SLAB.PTR
W9.01 BOOL  ; OPERATION.AUTO.CYCLE.RST.SLAB.PTR
W9.02 BOOL  ; OPERATION.AUTO.CYCLE.SLAB.PTR.CHNG
W9.03 BOOL  ; OPERATION.AUTO.CYCLE.BLOCK.POINTER.ENABLED
W9.04 BOOL  ; OPERATION.AUTO.CYCLE.INC.BLK.PTR
W9.05 BOOL  ; OPERATION.AUTO.cYCLE.DEC.BLK.PTR
W9.06 BOOL  ; OPERATION.AUTO.CYCLE.RST.BLK.PTR
W9.07 BOOL  ; OPERATION.AUTO.CYCLE.BLOCK.CHANGE
W9.08 BOOL  ; OPERATION.AUTO.CYCLE.BLOCK.COUNTED.EQUALS.BLOCK.QTY
W9.10 BOOL  ; OPERATION.AUTO.CYCLE.SEQUENCE.COMPLETE
BLADE_KERF D210 CHANNEL  ; BLADE.KERF.VALUE
BLADE_KERF_WORK_REAL D20 REAL  ; BLADE.KERF.VALUE.FLOAT.WORKING
BLK_DATA_END_ADR D1999 CHANNEL  ; Block Datat Tabe dimension end address
BLK_DATA_STRT_ADR D1000 CHANNEL  ; Dimension the Block Data Table - Start Address
BLK_DAT_RD_INIT H90.01 BOOL  ; Block Data Read Initiated
BLK_DAT_WRT_INIT H90.00 BOOL  ; Block Data Write Initiated
Block_Pointer Calculate_Pointer
CONST_MM_TO_INCH_DIV D7008 CHANNEL  ; CONST.MM.TO.INCH.DIVISOR
CUR_BLK_STORED_CRS_STP W332 CHANNEL  ; Current Block Stored Cross Stop Location
CUT_DEPTH D211 CHANNEL  ; CUT.DEPTH.VALUE.PROGRAMMED
CUT_DEPTH_VAL_FLT D22 REAL  ; CUT.DEPTH.VALUE.FLOAT
CUT_TRGT_CUR D212 CHANNEL  ; CUT.TARGET.CURRENT
DI_ENC_0_A 0.08 BOOL  ; _Ve
DI_ENC_0_B 0.09 BOOL  ; ENCODER.0.B
DI_ENC_0_Z 0.03 BOOL  ; ENCODER.0.Z
DI_ENC_1_A 0.06 BOOL  ; ENCODER.1.A
DI_ENC_1_B 0.07 BOOL  ; ENCODER.1.B
DI_ENC_1_Z 0.02 BOOL  ; ENCODER.1.Z
DI_FLOW_SW 1.00 BOOL  ; WATER.FLOW.SWITCH
DI_LONG_AXIS_HOME_SENS 1.01 BOOL  ; DI.LONG.AXIS.HOME.SENSOR
DI_LONG_AXIS_INDEX_CPT 0.04 BOOL  ; DI.LONG.AXIS.INDEX.COMPLETE
DI_LONG_MASTER_DRV_OK 0.10 BOOL  ; IO.LONG.AXIS.MASTER.DRIVE.OKAY.INPUT
DI_LONG_SLAVE_DRV_OK 0.01 BOOL  ; IO.LONG.SLAVE.DRIVE.OKAY.INPUT
DI_MCR_ON 0.00 BOOL  ; MCR.ON.POWER.ON
DI_SAFETY_ITLK 1.02 BOOL  ; SAFETY.GATE.INTERLOCK.INPUT
DI_SFT_STRT_FLT 0.11 BOOL  ; SAW.SOFT.START.FAULT
DI_TRANS_AXIS_DRV_OK 1.04 BOOL  ; IO.TRANSVERSE.AXIS.DRIVE.OKAY.INPUT
DI_TRANS_FWD 1.06 BOOL  ; TRANSVERSE.AXIS.FORWARD.LIMT.PROXIMITY
DI_TRANS_HOME 1.05 BOOL  ; TRANSVERSE.AXIS.HOME.PROXIMITY
DI_VERT_AXIS_DRV_OK 1.10 BOOL  ; IO.VERTICAL.AXIS.DRIVE.OKAY.INPUT
DI_VERT_FWD 1.08 BOOL  ; VERTICAL.AXIS.FORWARD.LIMIT
DI_VERT_HOME 1.07 BOOL  ; VERTICAL.AXIS.HOME.PROXIMITY
DO_ALARM_ANNUN 101.01 BOOL  ; ALARM.ANNUNCIATOR
DO_LAZER_ON 101.07 BOOL  ; LASER.ON
DO_LONG_AXIS_DRV_INDEX_CMD 101.02 BOOL  ; LONG.AXIS.MASTER.DRV.INDEX.COMMAND
DO_LONG_AXIS_HOME_INIT 101.06 BOOL  ; LONG.AXIS.MASTER.DRV.INITIATE.HOME.MOVE
DO_LONG_AXIS_JOG_LEFT 101.04 BOOL  ; LONG.AXIS.MASTER.DRV.JOG.LEFT
DO_LONG_AXIS_JOG_RIGHT 101.05 BOOL  ; LONG.AXIS.MASTER.DRV.JOG.RIGHT
DO_SFT_STRT_RUN 100.01 BOOL  ; SOFT.START.RUN
DO_SFT_STRT_STP 101.00 BOOL  ; SOFT.START.STOP
DO_TRANS_AXIS_FWD 100.04 BOOL  ; TRANSVERSE.AXIS.FORWARD
DO_TRANS_AXIS_REV 100.05 BOOL  ; TRANSVERSE.AXIS.REVERSE
DO_VERT_AXIS_BRK 101.03 BOOL  ; VERTICAL.AXIS.BRAKE.RELEASE
DO_VERT_AXIS_LWR 100.03 BOOL  ; VERTICAL.AXIS.LOWER
DO_VERT_AXIS_RAISE 100.02 BOOL  ; VERTICAL.AXIS.RAISE
DO_VERT_AXIS_SPD_SEL 100.06 BOOL  ; VERTICAL.AXIS.SPEED.SELECT.HIGH
DO_WATER_VLV 100.00 BOOL  ; WATER.VALVE
GLOBAL_HOME_REQUEST W0.15 BOOL  ; GLOBAL.HOME.REQUEST
HSC0_Init HSC0_INIT
HSC0_Init_Plx W0.00 BOOL  ; HSC0 Initialised at Power Up
HSC0_PWR_INIT H0.00 BOOL  ; HSC.0.PWR.INIT
HSC1_Init HSC1_INIT
HSC1_Init_Plx W1.00 BOOL  ; HSC1 Initialised at power up
HSC1_PWR_INIT H0.01 BOOL  ; HSC.1.PWR.INIT
IO_LAZER_PWR_OK H15.00 BOOL  ; IO.LAZER.POWER.OKAY
IO_LAZER_SG_OK H15.01 BOOL  ; IO.LAZER.SAFETY.GATE.OKAY
IO_SAW_NOT_SAFE_TO_RUN H13.03 BOOL  ; IO.SAW.NOT.SAFE.TO.RUN
IO_SAW_PWR_OK H13.00 BOOL  ; IO.SAW.POWER.OKAY
IO_SAW_SAFE_TO_RUN H13.02 BOOL  ; IO.SAW.SAFE.TO.RUN
IO_SAW_SG_OK H13.01 BOOL  ; IO.SAW.SAFETY.GATE.OKAY
IO_Saw_Safe_To_Run Op_2_State
IO_WTR_PWR_OK H14.00 BOOL  ; IO.WATER.POWER.OKAY
IO_WTR_SG_OK H14.01 BOOL  ; IO.WATER.SAFETY.GATE.OKAY
LAXISMFDBK A276 CHANNEL  ; LONG.AXIS.MASTER.FEEDBACK
MAIN_PWR_ERR W0.05 BOOL  ; MAIN.POWER.ERR
MC_AXIS_DRV_STP_STATE H11.12 BOOL  ; MC.VERTICAL.AXIS.DRIVE.STOP.STATE
MC_AXIS_LONG_FDBK D5000 WORD  ; MC.LONG.AXIS.FEEDBACK.LOW.WORD
MC_LONG_AXIS_AUTO_NOK H10.03 BOOL  ; MC.LONG.AXIS.AUTO.NOT.OKAY
MC_LONG_AXIS_AUTO_OK H10.02 BOOL  ; MC.LONG.AXIS.AUTO.OKAY
MC_LONG_AXIS_DRV_ACT 302.00 BOOL  ; MC.LONG.AXIS.DRIVE.ACTIVE
MC_LONG_AXIS_DRV_AT_ZERO 303.00 BOOL  ; MC.LONG.AXIS.DRIVE.AT.ZERO.SPEED
MC_LONG_AXIS_DRV_EN 304.00 BOOL  ; MC.LONG.AXIS.DRV.ENABLE
MC_LONG_AXIS_DRV_ERR H10.05 BOOL  ; MC.LONG.AXIS.DRIVE.ERROR
MC_LONG_AXIS_DRV_JOG_PLUS_INPUT_MON 324.00 BOOL  ; MC.LONG.AXIS.DRIVE.JOG.PLUS.INPUT.STATE.MONITOR
MC_LONG_AXIS_DRV_MAINS_LOSS 315.00 BOOL  ; MC.LONG.AXIS.MAINS.LOSS.FAULT
MC_LONG_AXIS_DRV_OK 301.00 BOOL  ; MC.LONG.AXIS.DRIVE.OKAY
MC_LONG_AXIS_DRV_OKAY H10.04 BOOL  ; MC.LONG.AXIS.DRIVE.OKAY
MC_LONG_AXIS_DRV_OL 317.00 BOOL  ; MC.LONG.AXIS.DRIVE.OVERLOAD.FAULT
MC_LONG_AXIS_DRV_RST 333.00 BOOL  ; MC.LONG.AXIS.DRIVE.RESET
MC_LONG_AXIS_DRV_RST_EN H10.11 BOOL  ; MC.LONG.AXIS.DRIVE.RESET.ENABLED
MC_LONG_AXIS_DRV_STOP_NOT 310.00 BOOL  ; MC.LONG.AXIS.DRIVE.STOP.NOT
MC_LONG_AXIS_DRV_UV 316.00 BOOL  ; MC.LONG.AXIS.DRIVE.BUS.UNDER.VOLTAGE.ERROR
MC_LONG_AXIS_DRV_WRN 319.00 BOOL  ; MC.LONG.AXIS.DRIVE.WARNING.[FAULT EXISTS]
MC_LONG_AXIS_ERR H10.14 BOOL  ; LONG.AXIS.ERROR.EXISTS
MC_LONG_AXIS_EZMTN_ERR 314 INT  ; MC.LONG.AXIS.DRIVE.EZMOTION.MODULE.ERROR
MC_LONG_AXIS_EZMTN_STATUS 312 LINT  ; MC.LONG.AXIS.DRIVE.EZMOTION.MODULE.STATUS
MC_LONG_AXIS_FDBK_REAL D5006 REAL  ; MC.LONG.AXIS.FEEDBACK.REAL
MC_LONG_AXIS_FDBK_REAL_SCALED D5010 REAL  ; MC.LONG.AXIS.FEEDBACK.SCALED
MC_LONG_AXIS_GATE_OK H10.01 BOOL  ; LONG.AXIS.SAFETY.GATE.OKAY
MC_LONG_AXIS_HOME_ACT H20.01 BOOL  ; MC.LONG.AXIS.HOMING.ACTIVE
MC_LONG_AXIS_HOME_CMD_INT H10.08 BOOL  ; MC.LONG.AXIS.HOME.COMMAND.INTERNAL
MC_LONG_AXIS_HOME_CMPLT H20.02 BOOL  ; MC.LONG.AXIS.HOMING.COMPLETED
MC_LONG_AXIS_HOME_EN H10.12 BOOL  ; MC.LONG.AXIS.HOME.INSTRUCTION.ENABLED
MC_LONG_AXIS_HOME_ERR H20.03 BOOL  ; MC.LONG.AXIS.HOMING.ERROR.OCCURED
MC_LONG_AXIS_HOME_INIT_MON 325.00 BOOL  ; MC.LONG.AXIS.HOME.INITIATE.INPUT.MONITOR
MC_LONG_AXIS_HOME_INIT_REQ H20.00 BOOL  ; MC.LONG.AXIS.HOME.INITIALISE.REQUEST
MC_LONG_AXIS_HOME_SENSOR_MON 326.00 BOOL  ; MC.LONG.AXIS.DRIVE.HOME.SENSOR.INPUT.MONITOR
MC_LONG_AXIS_JOGR_CMD H10.07 BOOL  ; MC.LONG.AXIS.JOG.RIGHT.COMMAND
MC_LONG_AXIS_JOG_ACT H10.09 BOOL  ; MC.LONG.AXIS.JOG.ACTIVE
MC_LONG_AXIS_JOG_EN H10.06 BOOL  ; MC.LONG.AXIS.JOG.ENABLED
MC_LONG_AXIS_JOG_ERR H10.10 BOOL  ; MC.LONG.AXIS.JOG.ERROR
MC_LONG_AXIS_JOG_MIN_INPUT_MON 323.00 BOOL  ; MC.LONG.AXIS.DRV.JOG.MINUS.INPUT.MONITOR
MC_LONG_AXIS_MIN_LIM_MON 321.00 BOOL  ; MC.LONG.AXIS.DRIVE.MINUS.LIMIT.ACTIVE.MONITOR
MC_LONG_AXIS_MODID 311 INT  ; MC.LONG.AXIS.DRIVE.EZMOTION.MODULE.ID
MC_LONG_AXIS_MOTION_CMD MC_Axis_Motion
MC_LONG_AXIS_PGM_INIT_MON 320.00 BOOL  ; MC.LONG.AXIS.DRIVE.EZMOTION.PROGRAM.INITIATE.MONITOR
MC_LONG_AXIS_PLUS_LIM_MON 322.00 BOOL  ; MC.LONG.AXIS.PLUS.LIMIT.ACTIVE.MONITOR
MC_LONG_AXIS_POS_REF_CMD_LOW D4 WORD  ; MC.LONG.AXIS.POSITION.REFERENCE.COMMAND.VALUE.LOW.WORD
MC_LONG_AXIS_PWR_OK H10.00 BOOL  ; LONG.AXIS.POWER.OKAY
MC_LONG_AXIS_RDY H10.15 BOOL  ; LONG.AXIS.MOTION.READY
MC_LONG_AXIS_RESET_CMD MC_Axis_Reset
MC_LONG_AXIS_TEMP_FLT 318.00 BOOL  ; MC.LONG.AXIS.DRIVE.OVER.TEMPERATURE.FAULT
MC_Long_Axis_Drv_OK Op_2_State
MC_Long_Axis_Home_Func MC_Axis_Srv_Home
MC_Op_Long_Axis_Jog MC_Axis_Jog
MC_Op_Trans_Axis_Jog_Cmd MC_Axis_Jog
MC_Op_Vert_Axis_Jog_Cmd MC_Axis_Jog
MC_PERM_TRANS_AXIS_AUTO_NOK H12.03 BOOL  ; MC.PERMISSIVE.TRANSVERSE.AXIS.AUTO.NOK
MC_PERM_TRANS_AXIS_AUTO_OK H12.02 BOOL  ; MC.PERMISSIVE.TRANSVERSE.AXIS.AUTO.OK
MC_TRANS_AXIS_DRV_ACT 402.00 BOOL  ; MC.TRANSVERSE.AXIS.DRIVE.ACTIVE
MC_TRANS_AXIS_DRV_AT_ZERO_SPD 403.00 BOOL  ; MC.TRANSVERSE.AXIS.DRIVE.AT.ZERO.SPEED
MC_TRANS_AXIS_DRV_ERR H12.05 BOOL  ; MC.TRANSVERSE.AXIS.DRIVE.ERROR
MC_TRANS_AXIS_DRV_GNRL_ERR 419.00 BOOL  ; MC.TRANSVERSE.AXIS.DRIVE.GENERAL.ERROR
MC_TRANS_AXIS_DRV_MAINS_LOSS 415.00 BOOL  ; MC.TRANSVERSE.AXIS.DRIVE.MAINS.LOSS
MC_TRANS_AXIS_DRV_NOT_STOP 410.00 BOOL  ; MC.TRANSVERSE.AXIS.DRIVE.NOT.STOP
MC_TRANS_AXIS_DRV_OK 401.00 BOOL  ; MC.TRANSVERSE.AXIS.DRIVE.OKAY.STATUS
MC_TRANS_AXIS_DRV_OK_PERM H12.04 BOOL  ; MC.PERMISSIVE.TRANSVERSE.AXIS.DRIVE.OKAY
MC_TRANS_AXIS_DRV_OL 417.00 BOOL  ; MC.TRANSVERSE.AXIS.DRIVE.OVERLOAD.ERROR
MC_TRANS_AXIS_DRV_PREC_REF_SEL 444.00 BOOL  ; MC.TRANSVERSE.AXIS.DRIVE.PRECISION.REFERENCE.SELECT
MC_TRANS_AXIS_DRV_RESET 433.00 BOOL  ; MC.TRANSVERSE.AXIS.DRIVE.ERROR.RESET
MC_TRANS_AXIS_DRV_RST MC_Axis_Reset
MC_TRANS_AXIS_DRV_RUN_FWD 405.00 BOOL  ; MC.TRANSVERSE.AXIS.DRIVE.RUN.FORWARD
MC_TRANS_AXIS_DRV_RUN_REV 407.00 BOOL  ; MC.TRANSVERSE.AXIS.DRIVE.RUN.REVERSE
MC_TRANS_AXIS_DRV_STP_STATE H12.12 BOOL  ; MC.TRANSVERSE.AXiS.DRIVE.STOP.STATE
MC_TRANS_AXIS_DRV_TEMP_ERR 418.00 BOOL  ; MC.TRANSVERSE.AXIS.DRIVE.TEMPERATURE.ERROR
MC_TRANS_AXIS_ERR H12.14 BOOL  ; TRANSVERSE.AXIS.ERROR.EXISTS
MC_TRANS_AXIS_FDBK_INTRM2 D28 LINT  ; MC.TRANSVERSE.AXIS.VELOCITY.FEEDBACK.INTERIM2
MC_TRANS_AXIS_FT_P_MIN D30 INT  ; MC.TRANSVERSE.AXIS.FEET.PER.MIN
MC_TRANS_AXIS_HOME_ACT H22.01 BOOL  ; MC.TRANSVERSE.AXIS.HOMING.ACTIVE
MC_TRANS_AXIS_HOME_CMP H22.02 BOOL  ; MC.TRANSVERSE.AXIS.HOMING.COMPLETED
MC_TRANS_AXIS_HOME_ERR H22.03 BOOL  ; MC.TRANSVERSE.AXIS.HOMING.ERROR
MC_TRANS_AXIS_HOME_INIT_REQ H22.00 BOOL  ; MC.TRANSVERSE.AXIS.HOME.INITIALISE.REQUEST
MC_TRANS_AXIS_JOG_ACT H12.09 BOOL  ; MC.TRANSVERSE.AXIS.JOG.COMMAND.ACTIVE
MC_TRANS_AXIS_JOG_CMD_ERR H12.10 BOOL  ; MC.TRANSVERSE.AXIS.JOG.COMMAND.ERROR
MC_TRANS_AXIS_JOG_EN H12.06 BOOL  ; MC.TRANSVERSE.AXIS.JOG.ENABLED
MC_TRANS_AXIS_JOG_FWD 406.00 BOOL  ; MC.TRANSVERSE.AXIS.DRIVE.JOG.FORWARD
MC_TRANS_AXIS_JOG_REV 408.00 BOOL  ; MC.TRANSVERSE.AXIS.DRIVE.JOG.REVERSE
MC_TRANS_AXIS_NOT_STP_MON H12.11 BOOL  ; MC.TRANSVERSE.AXIS.DRIVE.NOT.STOP.MONITOR
MC_TRANS_AXIS_PWR_OK H12.00 BOOL  ; TRANSVERSE.AXIS.POWER.OKAY
MC_TRANS_AXIS_READY H12.15 BOOL  ; MC.TRANSVERSE.READY
MC_TRANS_AXIS_SAFETY_GATE_OK H12.01 BOOL  ; TRANSVERSE.AXIS.SAFETY.GATE.OKAY
MC_TRANS_AXIS_VEL_FDBK_INTRM D26 LINT  ; MC.TRANSVERSE.AXIS.VELOCITY.FEEDBACK.INTERIM
MC_TRANS_MOTION_FOL_ERR MC_Axis_Motion_Monitor
MC_TRANS_POS_FDBK_SCALED D6010 REAL  ; MC.TRANSVERSE.AXIS.POSITION.FEEDBACK.INCHES.SCALED.REAL
MC_TRAN_AXIS_DRV_EN 404.00 BOOL  ; MC.TRANSVERSE.AXIS.DRIVE.ENABLE
MC_VERT_AXISDRV_NOT_STP 510.00 BOOL  ; MC.VERTICAL.AXIS.DRIVE.NOT.STOP
MC_VERT_AXIS_AUTO_OK H11.02 BOOL  ; MC.VERTICAL.AXIS.AUTO.OK
MC_VERT_AXIS_DRV_ACT 502.00 BOOL  ; MC.VERTICAL.AXIS.DRIVE.ACTIVE
MC_VERT_AXIS_DRV_AT_ZERO_SPD 503.00 BOOL  ; MC.VERTICAL.AXIS.DRIVE.AT.ZERO.SPEED
MC_VERT_AXIS_DRV_EN 504.00 BOOL  ; MC.VERTICAL.AXIS.DRIVE.ENABLE
MC_VERT_AXIS_DRV_ERR H11.05 BOOL  ; MC.VERTICAL.AXIS.DRIVE.ERROR
MC_VERT_AXIS_DRV_GNRL_ERR 519.00 BOOL  ; MC.VERTICAL.AXIS.DRIVE.GENERAL.ERROR
MC_VERT_AXIS_DRV_MAINS_LOSS 515.00 BOOL  ; MC.VERTICAL.AXIS.DRIVE.MAINS.LOSS
MC_VERT_AXIS_DRV_NOT_STP_MON H11.11 BOOL  ; MC.VERT.AXIS.DRV.NOT.STP.MON
MC_VERT_AXIS_DRV_OK 501.00 BOOL  ; MC.VERTICAL.AXIS.DRIVE.OKAY
MC_VERT_AXIS_DRV_OK_PERM H11.04 BOOL  ; MC.VERTICAL.AXIS.DRIVE.OKAY.PERMISSIVE
MC_VERT_AXIS_DRV_OL 517.00 BOOL  ; MC.VERTICAL.AXIS.DRIVE.OVERLOAD.ERROR
MC_VERT_AXIS_DRV_PREC_REF_SEL 544.00 BOOL  ; MC.VERTICAL.AXIS.DRIVE.PRECISION.REFERENCE.SELECT
MC_VERT_AXIS_DRV_RESET 533.00 BOOL  ; MC.VERTICAL.AXIS.DRIVE.RESET
MC_VERT_AXIS_DRV_RUN_REV 507.00 BOOL  ; MC.VERTICAL.AXIS.DRIVE.RUN.REVERSE
MC_VERT_AXIS_DRV_TEMP_ERR 518.00 BOOL  ; MC.VERTICAL.AXIS.DRIVE.TEMPERATURE.ERROR
MC_VERT_AXIS_ERR H11.14 BOOL  ; MC.VERTICAL.AXIS.ERROR
MC_VERT_AXIS_FDBK_BALLSC_REV_REAL D7004 CHANNEL  ; MC.VERTICAL.POSITION.FEEDBACK.BALLSCREW.REVOLUTIONS.REAL
MC_VERT_AXIS_FDBK_REAL_SCALED D7010 REAL  ; MC.VERTICAL.AXIS.FEEDBACK.REAL.SCALED.INCH
MC_VERT_AXIS_HOME_ACT H21.01 BOOL  ; MC.VERTICAL.AXIS.HOMING.ACTIVE
MC_VERT_AXIS_HOME_CMP H21.02 BOOL  ; MC.VERTICAL.AXIS.HOMING.COMPLETED
MC_VERT_AXIS_HOME_ERR H21.03 BOOL  ; MC.VERTICAL.AXIS.HOMING.ERROR
MC_VERT_AXIS_HOME_INIT_REQ H21.00 BOOL  ; MC.VERTICAL.AXIS.HOME.INITIALISE.REQUEST
MC_VERT_AXIS_JOG_ACT H11.09 BOOL  ; MC.VERTICAL.AXIS.JOG.ACTIVE
MC_VERT_AXIS_JOG_EN H11.06 BOOL  ; MC.VERTICAL.AXIS.JOG.ENABLED
MC_VERT_AXIS_JOG_FWD 506.00 BOOL  ; MC.VERTICAL.AXIS.DRIVE.JOG.FORWARD
MC_VERT_AXIS_JOG_REV 508.00 BOOL  ; MC.VERTICAL.AXIS.JOG.REVERSE
MC_VERT_AXIS_JO_CMD_ERR H11.10 BOOL  ; MC.VERTICAL.AXIS.JOG.COMMAND.ERROR
MC_VERT_AXIS_POS_FDBK_GB_SCALED_REAL D7002 CHANNEL  ; MC.VERTICAL.AXIS.POSITION.REVOLUTION.REAL
MC_VERT_AXIS_POS_FDBK_RAW D7000 CHANNEL  ; MC.VERTICAL.AXIS.POSITION.FEEDBACK.RAW.REAL
MC_VERT_AXIS_PWR_OK H11.00 BOOL  ; VERTICAL.AXIS.POWER.OKAY
MC_VERT_AXIS_RDY H11.15 BOOL  ; MC.VERTICAL.AXIS.READY
MC_VERT_AXIS_RST MC_Axis_Reset
MC_VERT_AXIS_RUN_FWD 505.00 BOOL  ; MC.VERTICAL.AXIS.DRIVE.RUN.FORWARD
MC_VERT_AXIS_SAFETY_GATE_OK H11.01 BOOL  ; VERTICAL.AXIS.SAFETY.GATE.OKAY
MC_VERT_MTN_FOLLOW_ERR MC_Axis_Motion_Monitor
MODE_AUTO_IND W130.14 BOOL  ; AUTOMATIC.MODE.INDICATOR
MODE_MAN_IND W130.13 BOOL  ; MANUAL.MODE.INDICATOR
MODE_SEL_AUTO W0.09 BOOL  ; MODE.SELECT.AUTOMATIC
MODE_SEL_AUTO_EN W0.11 BOOL  ; MODE.SELECT.AUTO.MODE.ENABLED
MODE_SEL_EN W0.07 BOOL  ; MODE.SELECT.ENABLED
MODE_SEL_MAN W0.08 BOOL  ; MODE.SELECT.MANUAL
MODE_SEL_MAN_EN W0.10 BOOL  ; MODE.SELECT.MANUAL.MODE.ENABLED
Message_Display Op_Message
Mode_Select Op_Mode_Sel
OI_ALARM_MESSAGE_SELECT Op_Message
OI_ALM_CLR W111 WORD  ; OI.ALARM.MESSAGE.COLOUR
OI_ALM_IND W130.15 BOOL  ; OI.ALARM.INDICATOR.ACTIVE
OI_ALM_SEL W110 WORD  ; OI.ALARM.MESSAGE.SELECT
OI_CTL_ALM_RESET W121.08 BOOL  ; OPERATION.CONTROL.ALARM.RESET.PB
OI_CTL_TRANS_AXIS_HOME_PB W120.12 BOOL  ; OI.TRANSVERSE.AXIS.HOME.PB
OI_CTL_WORD_1 W120 WORD  ; OI.CONTROL.WORD.1
OI_CTL_WORD_2 W121 WORD  ; OI.CONTROL.WORD.2
OI_CTRL_CYCLE_START W120.02 BOOL  ; OI.CONTROL.AUTOMATIC.CYCLE.START.PB
OI_CTRL_CYCLE_STOP_PB W120.01 BOOL  ; OI.CONTROL.AUTOMATIC.CYCLE.STOP.PB
OI_CTRL_H_A_SEL W120.00 BOOL  ; OI.CONTROL.HAND.AUTO.SELECTOR
OI_CTRL_MAC_STOP W120.03 BOOL  ; OI.CONTROL.AUTOMATIC.CYCLE.MACHINE.STOP
OI_HOME_ALL_PB W120.04 BOOL  ; OI.HOME.ALL.PB
OI_IND_WORD_1 W130 WORD  ; OI.INDICATE.WORD.1
OI_IND_WORD_2 W131 WORD  ; OI.INDICATE.WORD.2
OI_LONG_AXIS_HOME_REQ W121.01 BOOL  ; OI.LING.AXIS.HOME.REQUEST.PB
OI_LONG_AXIS_JOG_MINUS W120.15 BOOL  ; OI.LONG.AXIS.JOG.MINUS.PB
OI_LONG_AXIS_JOG_PLUS W121.00 BOOL  ; OI.LONG.AXIS.JOG.PLUS.PB
OI_MSG_CLR W101 INT  ; OI.MESSAGE.COLOUR
OI_MSG_SEL W100 INT  ; OI.MESSAGE.SELECT
OI_SAW_CUR_ACT_SCL D140 REAL  ; OI.SAW.CURRENT.SCALED
OI_SAW_CUR_CALC D120 REAL  ; OI.SCALING.SAW.CURRENT.PART1
OI_SAW_STP_PB W120.08 BOOL  ; OI.SAW.STOP.PB
OI_SAW_STRT_PB W120.07 BOOL  ; OI.SAW.START.PB
OI_SEQ_MSG_SEL W105 CHANNEL  ; OI.SEQUENCE.MESSAGE.SELECT
OI_SET_FIRST_CUT W121.06 BOOL  ; OI.SET.FIRST.CUT.REQUEST
OI_Saw_Mach_Stop Op_2_State
OI_TRANS_AXIS_JOG_HOME_PB W120.13 BOOL  ; OI.TRANSVERSE.AXIS.JOG.HOME.PB
OI_TRANS_AXIS_JO_FWD_PB W120.14 BOOL  ; OI.TRANSVERSE.AXIS.JOG.FORWARD.PB
OI_VERT_AXIS_JOG_FWD_PB W120.11 BOOL  ; OI.VERTICAL.AXIS.JOG.FORWARD.PB
OI_VERT_AXIS_JOG_HOME_PB W120.10 BOOL  ; OI.VERTICAL.AXIS.JOG.HOME.PB
OI_WTR_ON_SEL W120.06 BOOL  ; OI.WATER.ON.SELECTOR
OOI_LAZER_ON_SEL W120.05 BOOL  ; OI.LAZER.ON.SELECTOR
OPERATION_AUTO_CYC_INCREMENT_BLOCK Calculate_Pointer
OPERATION_AUTO_CYC_INCREMENT_SLAB Calculate_Pointer
OP_ALARM_RESET H0.13 BOOL  ; OPERATION.ALARM.RESET.REQUEST
OP_ALARM_STATE_ACTIVE H0.15 BOOL  ; OP.ALARM.STATE.ACTIVE(FAULTED)
OP_ALMS_RES_EN Op_2_State
OP_ALM_MON_EN H0.12 BOOL  ; OP.ALARM.MONITORING.ENABLED
OP_ALRM_MON_ACT H0.14 BOOL  ; OPERATION.ALARM.CONDITION.MONITRING.ACTIVE
OP_AUTO_BLK_ID D4114 INT  ; OPERATION.AUTO.CYCLE.BLOCK.ID
OP_AUTO_CYC_BLK_CNT D4102 INT  ; OPERATION.AUTO.CYCLE.BLOCK.ID
OP_AUTO_CYC_BLK_FCUT D4106 REAL  ; OPERATION.AUTO.CYCLE.BLOCK.FIRST.CUT.WORKING
OP_AUTO_CYC_BLK_HEIGHT D4100 REAL  ; OPERATION.AUTO.CYCLE.BLOCK.HEIGHT.WORKING
OP_AUTO_CYC_BLK_LEN D4104 REAL  ; OPERATION.AUTO.CYCLE.BLOCK.TRANSVERSE.AXIS.STOP.POSITION.WORKING
OP_AUTO_CYC_BLK_QTY D4116 INT  ; OPERATION.AUTO.CYCLE.BLOCK.QUANTITY
OP_AUTO_CYC_BLK_SLABQ D4108 INT  ; OPERATION.AUTO.CYCLE.CURRENT.BLOCK.SLAB.QUANTITY
OP_AUTO_CYC_CUR_BLK_1ST_CUT D106 REAL  ; Operation Auto Cycle Current Block First Cut Location
OP_AUTO_CYC_CUR_BLK_HGT D102 REAL  ; Operation Auto Cycle Current Block Height
OP_AUTO_CYC_CUR_BLK_ID D100 INT  ; Operation Auto Cycle Current Block ID
OP_AUTO_CYC_CUR_CRS_STP D104 REAL  ; Operation Auto ycle Current Block Cross Stop
OP_AUTO_CYC_CUR_NUM_BLKS D101 INT  ; Operation Auto Cycle Current Number of Blocks
OP_AUTO_CYC_CUR_NUM_SLABS D108 INT  ; Operation Auto Cycle Current Block Number of Blocks
OP_AUTO_CYC_CUR_SLAB_CUT_Q D111 INT  ; Operation Automatic Cycle Current Slab Cut Quantity
OP_AUTO_CYC_CUR_SLAB_ID D110 INT  ; Operation Automatic Cycle Current Slab ID
OP_AUTO_CYC_CUR_SLAB_SIZ D112 REAL  ; Operation Automatic Cycle Current Slab Size
OP_AUTO_CYC_SLAB_CUR_ID D4113 INT  ; OPERATION.AUTO.CYCLE.CURRENT.SLAB.ID
OP_AUTO_CYC_SLAB_CUT_QTY D4112 INT  ; OPERATION.AUTO.CYCLE.CURRENT.SLAB.CUT.QUANTITY
OP_AUTO_CYC_SLAB_SPARE D4118 INT  ; OPERATION.AUTO.CYCLE.SLAB.ID
OP_AUTO_CYC_SLAB_SZ D4110 REAL  ; OPERATION.AUTO.CYCLE.CURRENT.SLAB.SIZE
OP_Alarm_Monitor Op_Alarm_Monitor
OP_CTL_AUTO_CYCLE_RUN_STEP1 W6.03 BOOL  ; OP.CONTROL.AUTO.CYCLE.RUN.EXECUTE.STEP1
OP_CTL_AUTO_CYC_STRTUP_STATE W6.00 BOOL  ; OP.CONTROL.AUTO.CYCLE.START.STATE
OP_CTL_AUTO_CYC_STRT_SAW_RUN W6.01 BOOL  ; OP.CONTROL.AUTO.CYCLE.SAW.START.STEP.DONE
OP_CTL_AUTO_CYC_STRT_WATER_ON W6.02 BOOL  ; OP.CONTROL.AUTO.CYCLE.START.WATER.COMPLETE
OP_CTRL_LONG_AXIS_TARG_REAL D5100 REAL  ; Operatin Long Axis Target Real
OP_CUR_BLK_LAST_HGT W326 REAL  ; Current Block Last Block Height
OP_CUR_BLK_LST_1ST_CUT W334 REAL  ; Current Block Last First Cut Position
OP_CUR_BLK_LST_CRS_STP W330 REAL  ; Current Block Last Cross Stop Position
OP_CUR_BLK_SLAB_ID W338 INT  ; Current Block Last Slab ID
OP_CUR_BLK_STORED_HGT W328 REAL  ; Current Block Stored Block Height
OP_CUR_BLK_STORED_SLAB_ID W339 INT  ; Current Block Stored Slab ID
OP_CUR_BL_STORED_1ST_CUT W336 REAL  ; Current Block Stored First Cut Location
OP_CUR_SLAB_LAST_CUT_Q W340 INT  ; Current Slab Last cut quantity
OP_CUR_SLAB_LAST_SZ W342 REAL  ; Current Slab Last Cut Size
OP_CUR_SLAB_STORED_CUT_Q W341 INT  ; Current Slab Stored cut quantity
OP_CUR_SLAB_STORED_SIZE W344 REAL  ; Current Slab Stored Slab Size
OP_CYCLE_RUN Op_Cyc_Run
OP_CYCLE_START Op_Cyc_Strt
OP_CYC_STOP Op_Cyc_Stp
OP_FIRST_CYC_CMPLT H0.02 BOOL  ; FIRST.CYCLE.COMPLETED
OP_Mode_Indicator Op_Mode_Ind
OP_PGM_BLK_1ST_CUT W206 REAL  ; Current Programming Block First Cut Location
OP_PGM_CHK_BLK1_1ST_CUT D10006 REAL  ; Operation Program Check Block 1 First Cut
OP_PGM_CHK_BLK1_CRS_STP D10004 REAL  ; Operation Program Check Block 1 Cross Stop
OP_PGM_CHK_BLK1_HGT D1002 REAL  ; Operation Program Check Block1 Height
OP_PGM_CHK_BLK1_ID D10000 INT  ; Operation Program Check Block 1 Block ID
OP_PGM_CHK_BLK1_NUM_BLKS D10001 INT  ; Operation Program Check Block 1 Number of Blocks
OP_PGM_CHK_BLK1_NUM_SLABS D1008 INT  ; Operation Program Check Block 1 Number of Slabs
OP_PGM_CHK_BLK2_1ST_CUT D10016 REAL  ; Operation Program Check Block  First Cut
OP_PGM_CHK_BLK2_CRS_STP D10014 REAL  ; Operation Program Check Block 2 Cross Stop
OP_PGM_CHK_BLK2_HGT D10012 REAL  ; Operation Program Check Block2 Height
OP_PGM_CHK_BLK2_ID D10010 INT  ; Operation Program Check Block 2 Block ID
OP_PGM_CHK_BLK2_NUM_BLKS D10011 INT  ; Operation Program Check Block 2 Number of Blocks
OP_PGM_CHK_BLK2_NUM_SLABS D1018 INT  ; Operation Program Check Block 2 Number of Slabs
OP_PGM_CHK_BLK3_1ST_CUT D10026 REAL  ; Operation Program Check Block 3 First Cut
OP_PGM_CHK_BLK3_CRS_STP D10024 REAL  ; Operation Program Check Block 3 Cross Stop
OP_PGM_CHK_BLK3_HGT D10022 REAL  ; Operation Program Check Block3 Height
OP_PGM_CHK_BLK3_ID D10020 INT  ; Operation Program Check Block 3 Block ID
OP_PGM_CHK_BLK3_NUM_BLKS D10021 INT  ; Operation Program Check Block 3 Number of Blocks
OP_PGM_CHK_BLK3_NUM_SLABS D1028 INT  ; Operation Program Check Block 3 Number of Slabs
OP_PGM_CHK_BLK4_1ST_CUT D10036 REAL  ; Operation Program Check Block 4 First Cut
OP_PGM_CHK_BLK4_CRS_STP D10034 REAL  ; Operation Program Check Block 4 Cross Stop
OP_PGM_CHK_BLK4_HGT D10012 REAL  ; Operation Program Check Block 4 Height
OP_PGM_CHK_BLK4_ID D10030 INT  ; Operation Program Check Block 4 Block ID
OP_PGM_CHK_BLK4_NUM_BLKS D10031 INT  ; Operation Program Check Block 3 Number of Blocks
OP_PGM_CHK_BLK4_NUM_SLABS D1038 INT  ; Operation Program Check Block 4 Number of Slabs
OP_PGM_CHK_SLAB10_EN H25.09 BOOL  ; OPERATION.ENABLE.SLAB10.DISPLAY
OP_PGM_CHK_SLAB11_EN H25.10 BOOL  ; OPERATION.ENABLE.SLAB11.DISPLAY
OP_PGM_CHK_SLAB12_EN H25.11 BOOL  ; OPERATION.ENABLE.SLAB12.DISPLAY
OP_PGM_CHK_SLAB12_ID D12110 INT  ; Operation Program Check Slab 12 ID
OP_PGM_CHK_SLAB13_EN H25.12 BOOL  ; OPERATION.ENABLE.SLAB13.DISPLAY
OP_PGM_CHK_SLAB13_ID D12120 INT  ; Operation Program Check Slab 13 ID
OP_PGM_CHK_SLAB14_EN H25.13 BOOL  ; OPERATION.ENABLE.SLAB14.DISPLAY
OP_PGM_CHK_SLAB14_ID D12130 INT  ; Operation Program Check Slab 14 ID
OP_PGM_CHK_SLAB15_EN H25.14 BOOL  ; OPERATION.ENABLE.SLAB15.DISPLAY
OP_PGM_CHK_SLAB15_ID D12140 INT  ; Operation Program Check Slab 15 ID
OP_PGM_CHK_SLAB16_EN H25.15 BOOL  ; OPERATION.ENABLE.SLAB16.DISPLAY
OP_PGM_CHK_SLAB16_ID D12150 INT  ; Operation Program Check Slab 16 ID
OP_PGM_CHK_SLAB17_EN H26.00 BOOL  ; OPERATION.ENABLE.SLAB17.DISPLAY
OP_PGM_CHK_SLAB17_ID D21160 INT  ; Operation Program Check Slab 17 ID
OP_PGM_CHK_SLAB17_Q D12161 INT  ; Operation Program Check Slab 17 Quantity
OP_PGM_CHK_SLAB17_W D12162 REAL  ; Operation Program Check Slab 17 Size
OP_PGM_CHK_SLAB18_EN H26.01 BOOL  ; OPERATION.ENABLE.SLAB18.DISPLAY
OP_PGM_CHK_SLAB18_ID D12170 INT  ; Operation Program Check Slab 18 ID
OP_PGM_CHK_SLAB19_EN H26.02 BOOL  ; OPERATION.ENABLE.SLAB19.DISPLAY
OP_PGM_CHK_SLAB19_ID D12180 INT  ; Operation Program Check Slab 19 ID
OP_PGM_CHK_SLAB1_EN H25.00 BOOL  ; OPERATION.ENABLE.SLAB1.DISPLAY
OP_PGM_CHK_SLAB1_ID D11000 INT  ; Operation Program Check Slab 1 ID
OP_PGM_CHK_SLAB1_SZ D2002 REAL  ; Operation Program Check Slab 1 Size
OP_PGM_CHK_SLAB20_EN H26.03 BOOL  ; OPERATION.ENABLE.SLAB20.DISPLAY
OP_PGM_CHK_SLAB20_ID D12190 INT  ; Operation Program Check Slab 20 ID
OP_PGM_CHK_SLAB21_EN H26.04 BOOL  ; OPERATION.ENABLE.SLAB21.DISPLAY
OP_PGM_CHK_SLAB21_ID D12200 INT  ; Operation Program Check Slab 21 ID
OP_PGM_CHK_SLAB22_EN H26.05 BOOL  ; OPERATION.ENABLE.SLAB22.DISPLAY
OP_PGM_CHK_SLAB22_ID D12210 INT  ; Operation Program Check Slab 22 ID
OP_PGM_CHK_SLAB23_EN H26.06 BOOL  ; OPERATION.ENBLE.SLAB23.DISPLAY
OP_PGM_CHK_SLAB23_ID D12220 INT  ; Operation Program Check Slab 23 ID
OP_PGM_CHK_SLAB24_EN H26.07 BOOL  ; OPERATION.ENABLE.SLAB24.DISPLAY
OP_PGM_CHK_SLAB24_ID D12230 INT  ; Operation Program Check Slab 24 ID
OP_PGM_CHK_SLAB25_EN H26.08 BOOL  ; OPERATION.ENABLE.SLAB25.DISPLAY
OP_PGM_CHK_SLAB25_ID D12240 INT  ; Operation Program Check Slab 25 ID
OP_PGM_CHK_SLAB26_EN H26.09 BOOL  ; OPERATION.ENABLE.SLAB26.DISPLAY
OP_PGM_CHK_SLAB27_EN H26.10 BOOL  ; OPERATION.ENABLE.SLAB27.DISPLAY
OP_PGM_CHK_SLAB27_ID D12260 INT  ; Operation Program Check SLab 27 ID
OP_PGM_CHK_SLAB28_EN H26.11 BOOL  ; OPERATION.ENABLE.SLAB28.DISPLAY
OP_PGM_CHK_SLAB28_ID D12270 INT  ; Operation Program Check Slab 28 ID
OP_PGM_CHK_SLAB29_EN H26.12 BOOL  ; OPERATION.ENABLE.SLAB29.DISPLAY
OP_PGM_CHK_SLAB29_ID D12280 INT  ; Operation Program Check Slab 29 ID
OP_PGM_CHK_SLAB2_C_Q D11011 INT  ; Operation Program Check Slab2 Cut Quantity
OP_PGM_CHK_SLAB2_EN H25.01 BOOL  ; OPERATION.ENABLE.SLAB2.DISPLAY
OP_PGM_CHK_SLAB2_ID D11010 INT  ; Operation Program Check Block1 Slab 2 ID
OP_PGM_CHK_SLAB2_SZ D11012 REAL  ; Operation Program Check Slab 2 Size
OP_PGM_CHK_SLAB30_EN H26.13 BOOL  ; OPERATIOn.ENABLE.SLAB30.DISPLAY
OP_PGM_CHK_SLAB30_ID D12290 INT  ; Operation Program Check Slab 30 ID
OP_PGM_CHK_SLAB31_EN H26.14 BOOL  ; Operation Enable Slab 31 Display
OP_PGM_CHK_SLAB32_EN H26.15 BOOL  ; Operation Program Check Slab 32 Display
OP_PGM_CHK_SLAB33_EN H27.00 BOOL  ; Operation Program Check Slab 33 Enable Display
OP_PGM_CHK_SLAB34_EN H27.01 BOOL  ; Operation Program Check Slab34 Enable Display
OP_PGM_CHK_SLAB35_EN H27.02 BOOL
OP_PGM_CHK_SLAB36_EN H27.03 BOOL
OP_PGM_CHK_SLAB37_EN H27.04 BOOL
OP_PGM_CHK_SLAB39_EN H27.06 BOOL
OP_PGM_CHK_SLAB3_C_Q D11021 INT  ; Operation Program Check Slab 3 Cut Quantity
OP_PGM_CHK_SLAB3_EN H25.02 BOOL  ; OPERATION.ENABLE.SLAB3.DISPLAY
OP_PGM_CHK_SLAB3_ID D11020 INT  ; Operation Program Check Slab 3 ID
OP_PGM_CHK_SLAB3_SZ D11022 REAL  ; Operation Program Check Slab 3 Size
OP_PGM_CHK_SLAB40_EN H27.07 BOOL
OP_PGM_CHK_SLAB41_EN H27.08 BOOL
OP_PGM_CHK_SLAB42_EN H27.09 BOOL
OP_PGM_CHK_SLAB43_EN H27.10 BOOL
OP_PGM_CHK_SLAB44_EN H27.11 BOOL
OP_PGM_CHK_SLAB45_EN H27.12 BOOL
OP_PGM_CHK_SLAB46_EN H27.13 BOOL
OP_PGM_CHK_SLAB47_EN H27.14 BOOL
OP_PGM_CHK_SLAB48_EN H27.15 BOOL
OP_PGM_CHK_SLAB49_EN H28.00 BOOL
OP_PGM_CHK_SLAB4_C_Q D11031 INT  ; Operation Program Check Slab 4 Cut Quantity
OP_PGM_CHK_SLAB4_EN H25.03 BOOL  ; OPERATION.ENABLE.SLAB4.DISPLAY
OP_PGM_CHK_SLAB4_ID D11030 INT  ; Operation Program Check Slab 4 ID
OP_PGM_CHK_SLAB4_SZ D11032 REAL  ; Operation Program Check Slab 4 Size
OP_PGM_CHK_SLAB50_EN H28.01 BOOL
OP_PGM_CHK_SLAB51_EN H28.02 BOOL  ; Operation Program Check Slab 51 Enable Display
OP_PGM_CHK_SLAB52_EN H28.03 BOOL
OP_PGM_CHK_SLAB53_EN H28.04 BOOL
OP_PGM_CHK_SLAB54_EN H28.05 BOOL
OP_PGM_CHK_SLAB55_EN H28.06 BOOL
OP_PGM_CHK_SLAB56_EN H28.07 BOOL
OP_PGM_CHK_SLAB57_EN H28.08 BOOL
OP_PGM_CHK_SLAB58_EN H28.09 BOOL
OP_PGM_CHK_SLAB59_EN H28.10 BOOL
OP_PGM_CHK_SLAB5_EN H25.04 BOOL  ; OPERATION.ENABLE.SLAB5.DISPLAY
OP_PGM_CHK_SLAB60_EN H28.11 BOOL
OP_PGM_CHK_SLAB61_EN H28.12 BOOL
OP_PGM_CHK_SLAB62_EN H28.13 BOOL
OP_PGM_CHK_SLAB63_EN H28.14 BOOL
OP_PGM_CHK_SLAB64_EN H28.15 BOOL
OP_PGM_CHK_SLAB65_EN H29.00 BOOL
OP_PGM_CHK_SLAB66_EN H29.01 BOOL
OP_PGM_CHK_SLAB67_EN H29.02 BOOL
OP_PGM_CHK_SLAB68_EN H29.03 BOOL
OP_PGM_CHK_SLAB69_EN H29.04 BOOL
OP_PGM_CHK_SLAB6_EN H25.05 BOOL  ; OPERATION.ENABLE.SLAB6.DISPLAY
OP_PGM_CHK_SLAB70_EN H29.05 BOOL
OP_PGM_CHK_SLAB71_EN H29.06 BOOL
OP_PGM_CHK_SLAB72_EN H29.07 BOOL
OP_PGM_CHK_SLAB73_EN H29.08 BOOL
OP_PGM_CHK_SLAB74_EN H29.09 BOOL
OP_PGM_CHK_SLAB75_EN H29.10 BOOL
OP_PGM_CHK_SLAB76_EN H29.11 BOOL
OP_PGM_CHK_SLAB77_EN H29.12 BOOL
OP_PGM_CHK_SLAB78_EN H29.13 BOOL
OP_PGM_CHK_SLAB79_EN H29.14 BOOL
OP_PGM_CHK_SLAB7_EN H25.06 BOOL  ; OPERATION.ENABLE.SLAB7.DISPLAY
OP_PGM_CHK_SLAB80_EN H29.15 BOOL
OP_PGM_CHK_SLAB81_EN H30.00 BOOL
OP_PGM_CHK_SLAB82_EN H30.01 BOOL
OP_PGM_CHK_SLAB83_EN H30.02 BOOL
OP_PGM_CHK_SLAB8_EN H25.07 BOOL  ; OPERATION.ENABLE.SLAB8.DISPLAY
OP_PGM_CHK_SLAB9_EN H25.08 BOOL  ; OERATION.ENABLE.SLAB9.DISPLAY
OP_PGM_CHK_SLAB_26_ID D12250 INT  ; Operation Program Check Slab 26 ID
OP_PGM_CHK_SLAB_38_EN H27.05 BOOL
OP_PGM_CHK_SLAB_C_Q D11001 INT  ; Operation Program Check Slab1 Cut Quantity
OP_PGM_CUR_BLK_CRS_STP W204 REAL  ; Current Programming Block Cross Stop Location
OP_PGM_CUR_BLK_HT W202 REAL  ; Current Programming Block Height
OP_PGM_CUR_BLK_SLAB_CNT W208 INT  ; Current Block Programmed Slab Count
OP_PGM_CUR_SLAB_ID W210 INT  ; Current Programming Slab ID
OP_PGM_CUR_SLAB_QTY W211 INT  ; Current Slab Programmed Quantity to cut
OP_PGM_CUR_SLAB_SZ W212 REAL  ; OPERATION.CURRENT.SLAB.SIZE.REAL
OP_PRG_CHK_SLAB10_CUT_Q D12091 INT  ; Operation Program Check Slab 10 Cut Quantity
OP_PRG_CHK_SLAB10_ID D12090 INT  ; Operation Program Check Slab 10 ID
OP_PRG_CHK_SLAB10_W D12092 REAL  ; Operation Program Check Slab 10 Width
OP_PRG_CHK_SLAB11_ID D12100 INT  ; Operation Prgoram Check Slab 11 ID
OP_PRG_CHK_SLAB1_CUT_Q D12001 INT  ; Operation Program Check Slab 1 Cut Quantity
OP_PRG_CHK_SLAB1_ID D12000 INT  ; Operation Program Check Slab 1 ID
OP_PRG_CHK_SLAB1_W D12002 REAL  ; Operation Program Check Slab 1 Width
OP_PRG_CHK_SLAB2_CUT_Q D12011 INT  ; Operation Program Check Slab 2 Cut Quantity
OP_PRG_CHK_SLAB2_ID D12010 INT  ; Operation Program Check Slab 2 ID
OP_PRG_CHK_SLAB2_W D12012 REAL  ; Operation Program Check Slab 2 Width
OP_PRG_CHK_SLAB3_CUT_Q D12021 INT  ; Operation Program Check Slab 3 Cut Quantity
OP_PRG_CHK_SLAB3_ID D12020 INT  ; Operation Program Check Slab 3 ID
OP_PRG_CHK_SLAB3_W D12022 REAL  ; Operation Program Check Slab 3 Width
OP_PRG_CHK_SLAB4_CUT_Q D12031 INT  ; Operation Program Check Slab 4 Cut Quantity
OP_PRG_CHK_SLAB4_ID D12030 INT  ; Operation Program Check Slab 4 ID
OP_PRG_CHK_SLAB4_W D12032 REAL  ; Operation Program Check Slab 4 Width
OP_PRG_CHK_SLAB5_CUT_Q D12041 INT  ; Operation Program Check Slab 5 Cut Quantity
OP_PRG_CHK_SLAB5_ID D12040 INT  ; Operation Program Check Slab 5 ID
OP_PRG_CHK_SLAB5_W D12042 REAL  ; Operation Program Check Slab 5 Width
OP_PRG_CHK_SLAB6_CUT_Q D12051 INT  ; Operation Program Check Slab 6 Cut Quantity
OP_PRG_CHK_SLAB6_ID D12050 INT  ; Operation Program Check Slab 6 ID
OP_PRG_CHK_SLAB6_W D12052 REAL  ; Operation Program Check Slab 6 Width
OP_PRG_CHK_SLAB7_CUT_Q D12061 INT  ; Operation Program Check Slab 7 Cut Quantity
OP_PRG_CHK_SLAB7_ID D12060 INT  ; Operation Program Check Slab 7 ID
OP_PRG_CHK_SLAB7_W D12062 REAL  ; Operation Program Check Slab 7 Width
OP_PRG_CHK_SLAB8_CUT_Q D12071 INT  ; Operation Program Check Slab 8 Cut Quantity
OP_PRG_CHK_SLAB8_ID D12070 INT  ; Operation Program Check Slab 8 ID
OP_PRG_CHK_SLAB9_CUT_Q D12081 INT  ; Operation Program Check Slab 9 Cut Quantity
OP_PRG_CHK_SLAB9_ID D12080 INT  ; Operation Program Check Slab 9 ID
OP_PRG_CHK_SLAB9_W D12082 REAL  ; Operation Program Check Slab 9 Width
OP_PRG_CHK_SLAB_W D12072 REAL  ; Operation Program Check Slab 8 Width
OP_Power_On_Check Op_2_State
OP_SAW_CUR_INT_CALC D122 REAL  ; OPERATION.SAW.CURRENT.INTERNAL
OP_SEQUENCE_STATE Op_Sequence_Step_State_Validate
OP_STEP_ENGINE Op_Cycle_Step
Op_Gate_Monitor Op_2_State
Op_Long_Axis_Mach_Stop Op_2_State
Op_Mach_Stop_Water Op_2_State
Op_Perm_Long_Auto Op_2_State
Op_Trans_Auto_Ok Op_2_State
Op_Trans_Axis_Drv_Ok Op_2_State
Op_Trans_Axis_Mach_Stop Op_2_State
Op_Vert_Auto_Ok Op_2_State
Op_Vert_Axis_Mach_Stop Op_2_State
Op_Vert_Axis_Ok Op_2_State
POWER_ON W0.03 BOOL  ; POWER.ON.MAIN
SAFETY_GATE_ERR W0.06 BOOL  ; SAFETY.GATE.ERR
SAFETY_GATE_OK W0.04 BOOL  ; SAFETY.GATE.OKAY
SLAB_DATA_END_ADR D2999 CHANNEL  ; DIMENSION.SLAB.DATA.TABLE.END.ADDRESS
SLAB_DATA_START_ADR D2000 CHANNEL  ; DIMENSION.SLAB.DATA.TABLE.START.ADDRESS
Slab_Pointer Calculate_Pointer
TARGET_CURRENT_WKNG D24 REAL  ; TARGET.CURRENT.WORKING.FLOAT
TRANS_POS_FDBK A272 CHANNEL  ; TRANSVERSE.POSITION.FEEDBACK.RAW
VERT_POS_FDBK A270 CHANNEL  ; VERTICAL.POSITION.FEEDBACK.RAW

## Program Main (cyclic task 0)
; Main saw program file

### Section Init_HSC

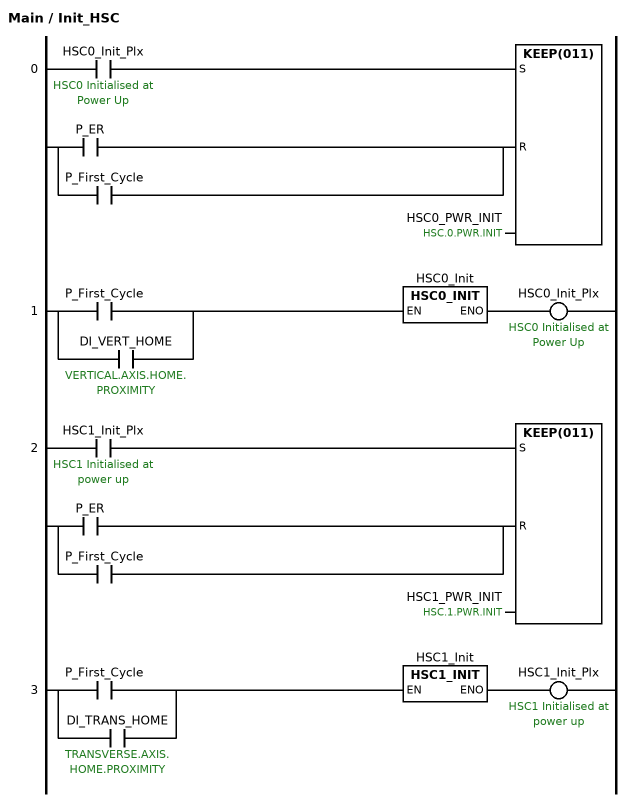
; rung 0
LD HSC0_Init_Plx  ; HSC0 Initialised at Power Up
LD P_ER
OR P_First_Cycle
KEEP(011) HSC0_PWR_INIT  ; HSC.0.PWR.INIT
; rung 1
LD P_First_Cycle
OR DI_VERT_HOME  ; VERTICAL.AXIS.HOME.PROXIMITY
CALL HSC0_Init : HSC0_INIT ()
OUT HSC0_Init_Plx  ; HSC0 Initialised at Power Up
; rung 2
LD HSC1_Init_Plx  ; HSC1 Initialised at power up
LD P_ER
OR P_First_Cycle
KEEP(011) HSC1_PWR_INIT  ; HSC.1.PWR.INIT
; rung 3
LD P_First_Cycle
OR DI_TRANS_HOME  ; TRANSVERSE.AXIS.HOME.PROXIMITY
CALL HSC1_Init : HSC1_INIT ()
OUT HSC1_Init_Plx  ; HSC1 Initialised at power up

### Section Interlock_Alarm

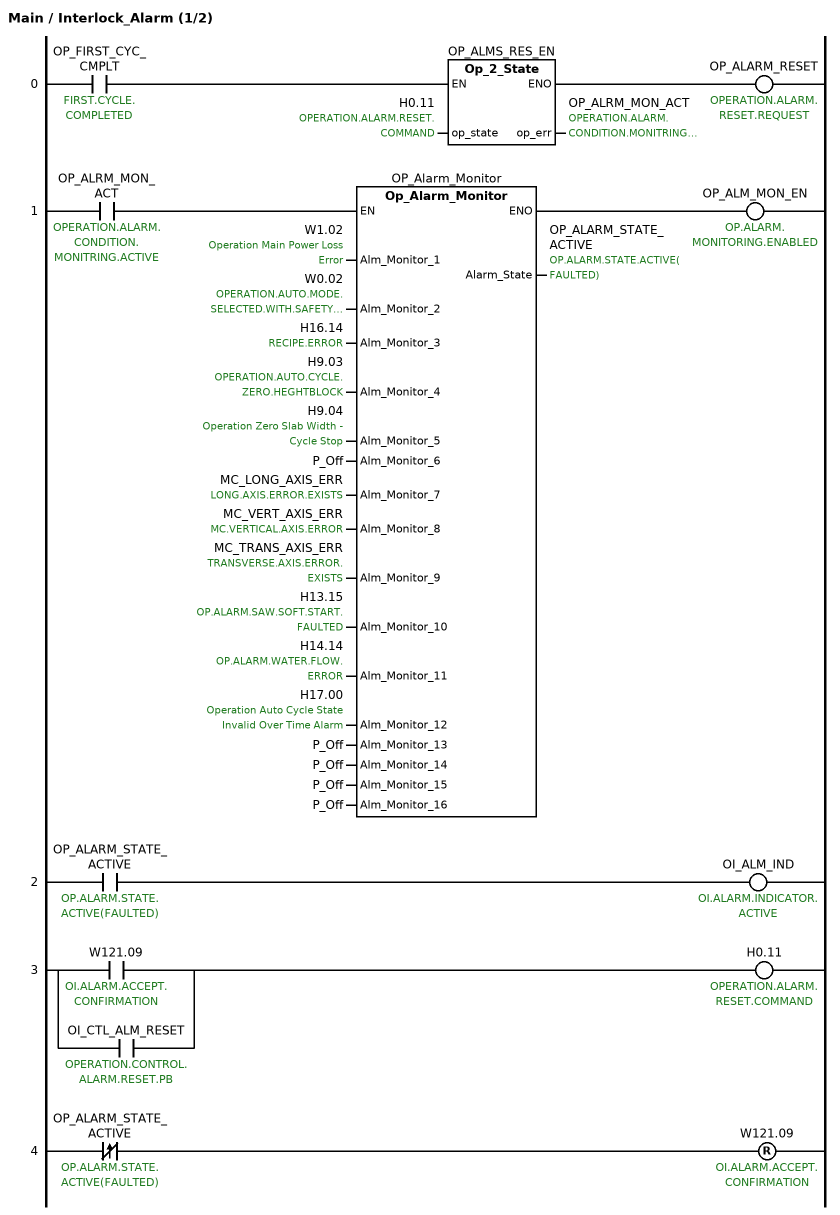
; rung 0
LD OP_FIRST_CYC_CMPLT  ; FIRST.CYCLE.COMPLETED
CALL OP_ALMS_RES_EN : Op_2_State (op_state := H0.11, op_err => OP_ALRM_MON_ACT)  ; OPERATION.ALARM.RESET.COMMAND, OPERATION.ALARM.CONDITION.MONITRING.ACTIVE
OUT OP_ALARM_RESET  ; OPERATION.ALARM.RESET.REQUEST
; rung 1
LD OP_ALRM_MON_ACT  ; OPERATION.ALARM.CONDITION.MONITRING.ACTIVE
CALL OP_Alarm_Monitor : Op_Alarm_Monitor (Alm_Monitor_1 := W1.02, Alm_Monitor_2 := W0.02, Alm_Monitor_3 := H16.14, Alm_Monitor_4 := H9.03, Alm_Monitor_5 := H9.04, Alm_Monitor_6 := P_Off, Alm_Monitor_7 := MC_LONG_AXIS_ERR, Alm_Monitor_8 := MC_VERT_AXIS_ERR, Alm_Monitor_9 := MC_TRANS_AXIS_ERR, Alm_Monitor_10 := H13.15, Alm_Monitor_11 := H14.14, Alm_Monitor_12 := H17.00, Alm_Monitor_13 := P_Off, Alm_Monitor_14 := P_Off, Alm_Monitor_15 := P_Off, Alm_Monitor_16 := P_Off, Alarm_State => OP_ALARM_STATE_ACTIVE)  ; Operation Main Power Loss Error, OPERATION.AUTO.MODE.SELECTED.WITH.SAFETY.GATE.OPEN, RECIPE.ERROR, OPERATION.AUTO.CYCLE.ZERO.HEGHTBLOCK, Operation Zero Slab Width - Cycle Stop, LONG.AXIS.ERROR.EXISTS, MC.VERTICAL.AXIS.ERROR, TRANSVERSE.AXIS.ERROR.EXISTS, OP.ALARM.SAW.SOFT.START.FAULTED, OP.ALARM.WATER.FLOW.ERROR, Operation Auto Cycle State Invalid Over Time Alarm, OP.ALARM.STATE.ACTIVE(FAULTED)
OUT OP_ALM_MON_EN  ; OP.ALARM.MONITORING.ENABLED
; rung 2
LD OP_ALARM_STATE_ACTIVE  ; OP.ALARM.STATE.ACTIVE(FAULTED)
OUT OI_ALM_IND  ; OI.ALARM.INDICATOR.ACTIVE
; rung 3
LD W121.09  ; OI.ALARM.ACCEPT.CONFIRMATION
OR OI_CTL_ALM_RESET  ; OPERATION.CONTROL.ALARM.RESET.PB
OUT H0.11  ; OPERATION.ALARM.RESET.COMMAND
; rung 4
@LDNOT OP_ALARM_STATE_ACTIVE  ; OP.ALARM.STATE.ACTIVE(FAULTED)
RSET W121.09  ; OI.ALARM.ACCEPT.CONFIRMATION

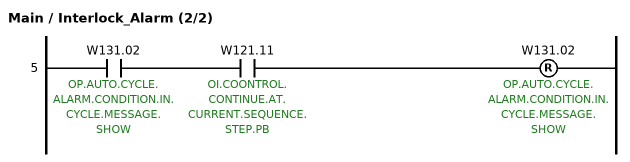
; rung 5
LD W131.02  ; OP.AUTO.CYCLE.ALARM.CONDITION.IN.CYCLE.MESSAGE.SHOW
AND W121.11  ; OI.COONTROL.CONTINUE.AT.CURRENT.SEQUENCE.STEP.PB
RSET W131.02  ; OP.AUTO.CYCLE.ALARM.CONDITION.IN.CYCLE.MESSAGE.SHOW

### Section Ctl_Power

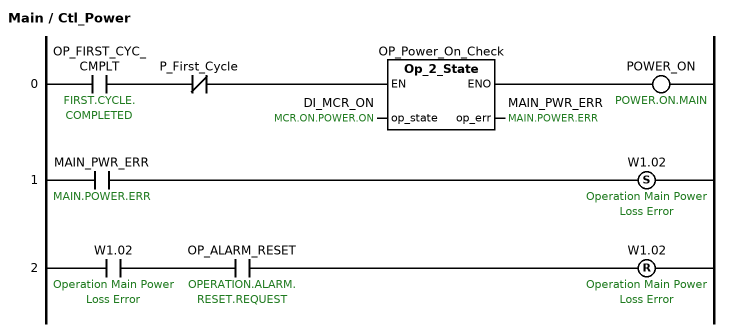
; rung 0
LD OP_FIRST_CYC_CMPLT  ; FIRST.CYCLE.COMPLETED
ANDNOT P_First_Cycle
CALL OP_Power_On_Check : Op_2_State (op_state := DI_MCR_ON, op_err => MAIN_PWR_ERR)  ; MCR.ON.POWER.ON, MAIN.POWER.ERR
OUT POWER_ON  ; POWER.ON.MAIN
; rung 1
LD MAIN_PWR_ERR  ; MAIN.POWER.ERR
SET W1.02  ; Operation Main Power Loss Error
; rung 2
LD W1.02  ; Operation Main Power Loss Error
AND OP_ALARM_RESET  ; OPERATION.ALARM.RESET.REQUEST
RSET W1.02  ; Operation Main Power Loss Error

### Section Ctl_Safety

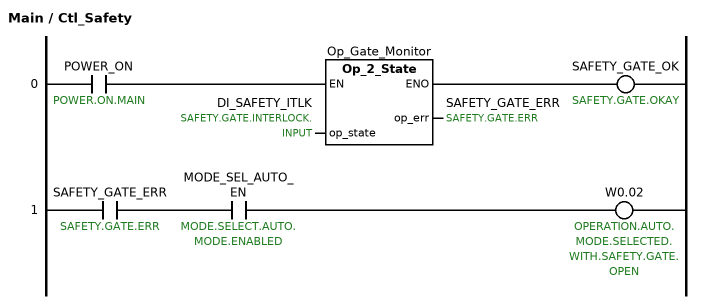
; rung 0
LD POWER_ON  ; POWER.ON.MAIN
CALL Op_Gate_Monitor : Op_2_State (op_state := DI_SAFETY_ITLK, op_err => SAFETY_GATE_ERR)  ; SAFETY.GATE.INTERLOCK.INPUT, SAFETY.GATE.ERR
OUT SAFETY_GATE_OK  ; SAFETY.GATE.OKAY
; rung 1
LD SAFETY_GATE_ERR  ; SAFETY.GATE.ERR
AND MODE_SEL_AUTO_EN  ; MODE.SELECT.AUTO.MODE.ENABLED
OUT W0.02  ; OPERATION.AUTO.MODE.SELECTED.WITH.SAFETY.GATE.OPEN

### Section Ctl_Mode

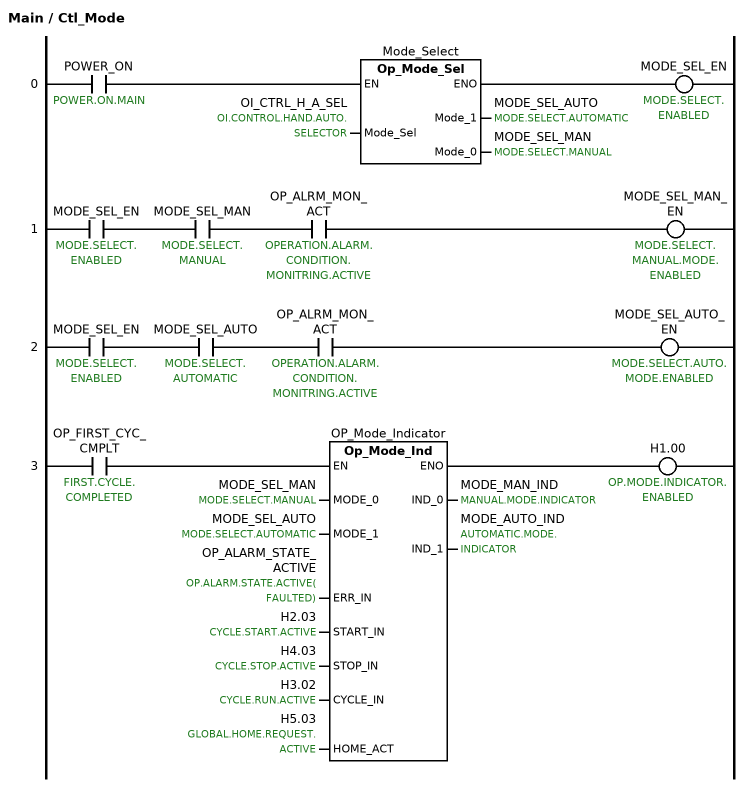
; rung 0
LD POWER_ON  ; POWER.ON.MAIN
CALL Mode_Select : Op_Mode_Sel (Mode_Sel := OI_CTRL_H_A_SEL, Mode_1 => MODE_SEL_AUTO, Mode_0 => MODE_SEL_MAN)  ; OI.CONTROL.HAND.AUTO.SELECTOR, MODE.SELECT.AUTOMATIC, MODE.SELECT.MANUAL
OUT MODE_SEL_EN  ; MODE.SELECT.ENABLED
; rung 1
LD MODE_SEL_EN  ; MODE.SELECT.ENABLED
AND MODE_SEL_MAN  ; MODE.SELECT.MANUAL
AND OP_ALRM_MON_ACT  ; OPERATION.ALARM.CONDITION.MONITRING.ACTIVE
OUT MODE_SEL_MAN_EN  ; MODE.SELECT.MANUAL.MODE.ENABLED
; rung 2
LD MODE_SEL_EN  ; MODE.SELECT.ENABLED
AND MODE_SEL_AUTO  ; MODE.SELECT.AUTOMATIC
AND OP_ALRM_MON_ACT  ; OPERATION.ALARM.CONDITION.MONITRING.ACTIVE
OUT MODE_SEL_AUTO_EN  ; MODE.SELECT.AUTO.MODE.ENABLED
; rung 3
LD OP_FIRST_CYC_CMPLT  ; FIRST.CYCLE.COMPLETED
CALL OP_Mode_Indicator : Op_Mode_Ind (MODE_0 := MODE_SEL_MAN, MODE_1 := MODE_SEL_AUTO, ERR_IN := OP_ALARM_STATE_ACTIVE, START_IN := H2.03, STOP_IN := H4.03, CYCLE_IN := H3.02, HOME_ACT := H5.03, IND_0 => MODE_MAN_IND, IND_1 => MODE_AUTO_IND)  ; MODE.SELECT.MANUAL, MODE.SELECT.AUTOMATIC, OP.ALARM.STATE.ACTIVE(FAULTED), CYCLE.START.ACTIVE, CYCLE.STOP.ACTIVE, CYCLE.RUN.ACTIVE, GLOBAL.HOME.REQUEST.ACTIVE, MANUAL.MODE.INDICATOR, AUTOMATIC.MODE.INDICATOR
OUT H1.00  ; OP.MODE.INDICATOR.ENABLED

### Section Ctl_Cycle_Start

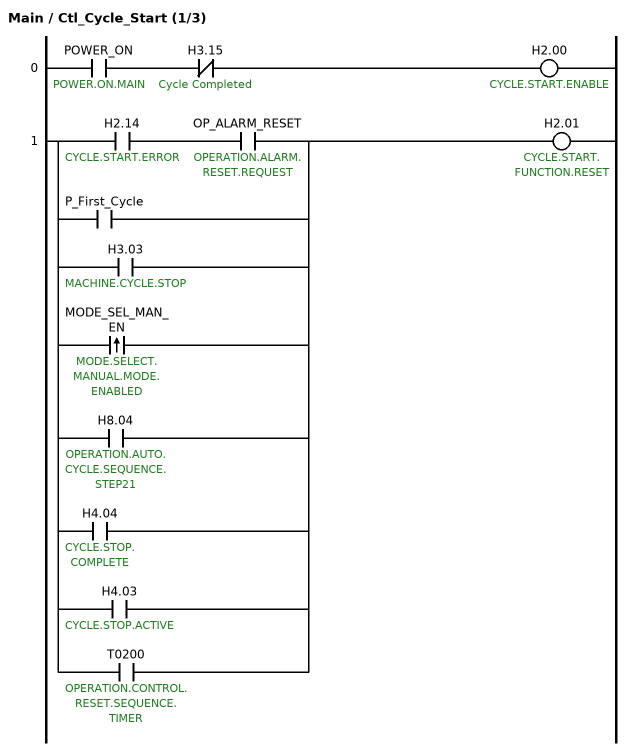
; rung 0
LD POWER_ON  ; POWER.ON.MAIN
ANDNOT H3.15  ; Cycle Completed
OUT H2.00  ; CYCLE.START.ENABLE
; rung 1
LD H2.14  ; CYCLE.START.ERROR
AND OP_ALARM_RESET  ; OPERATION.ALARM.RESET.REQUEST
OR P_First_Cycle
OR H3.03  ; MACHINE.CYCLE.STOP
@OR MODE_SEL_MAN_EN  ; MODE.SELECT.MANUAL.MODE.ENABLED
OR H8.04  ; OPERATION.AUTO.CYCLE.SEQUENCE.STEP21
OR H4.04  ; CYCLE.STOP.COMPLETE
OR H4.03  ; CYCLE.STOP.ACTIVE
OR T0200  ; OPERATION.CONTROL.RESET.SEQUENCE.TIMER
OUT H2.01  ; CYCLE.START.FUNCTION.RESET

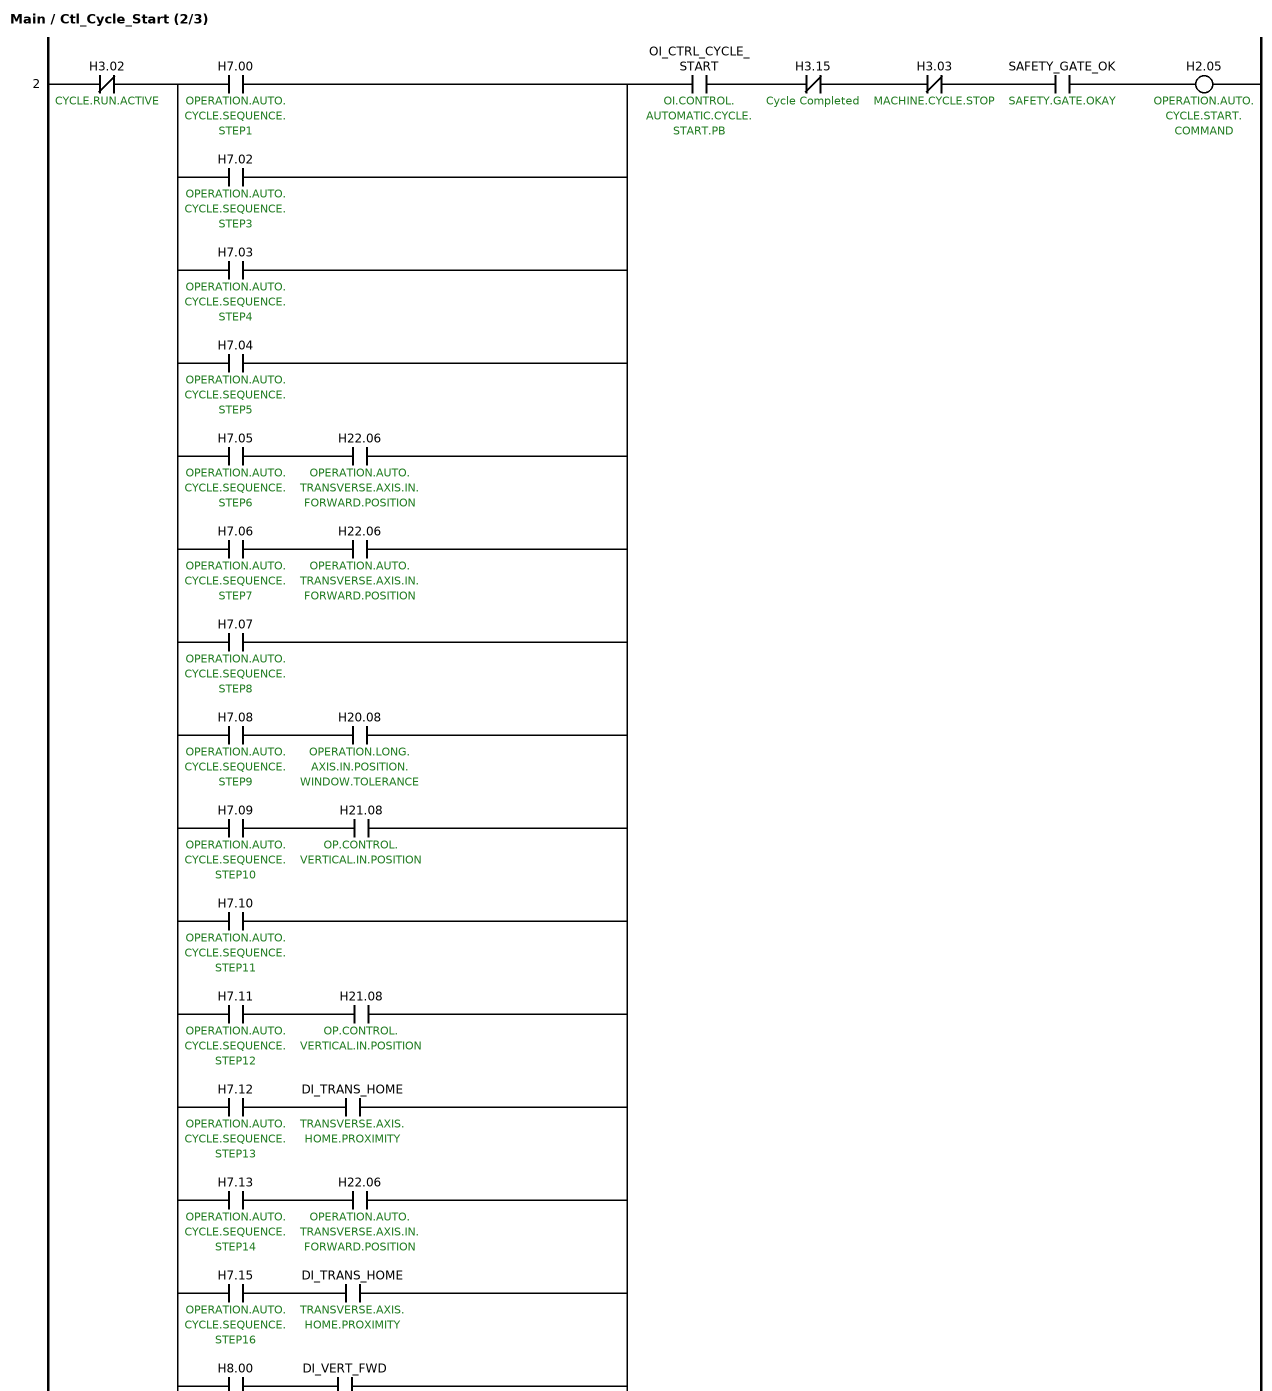

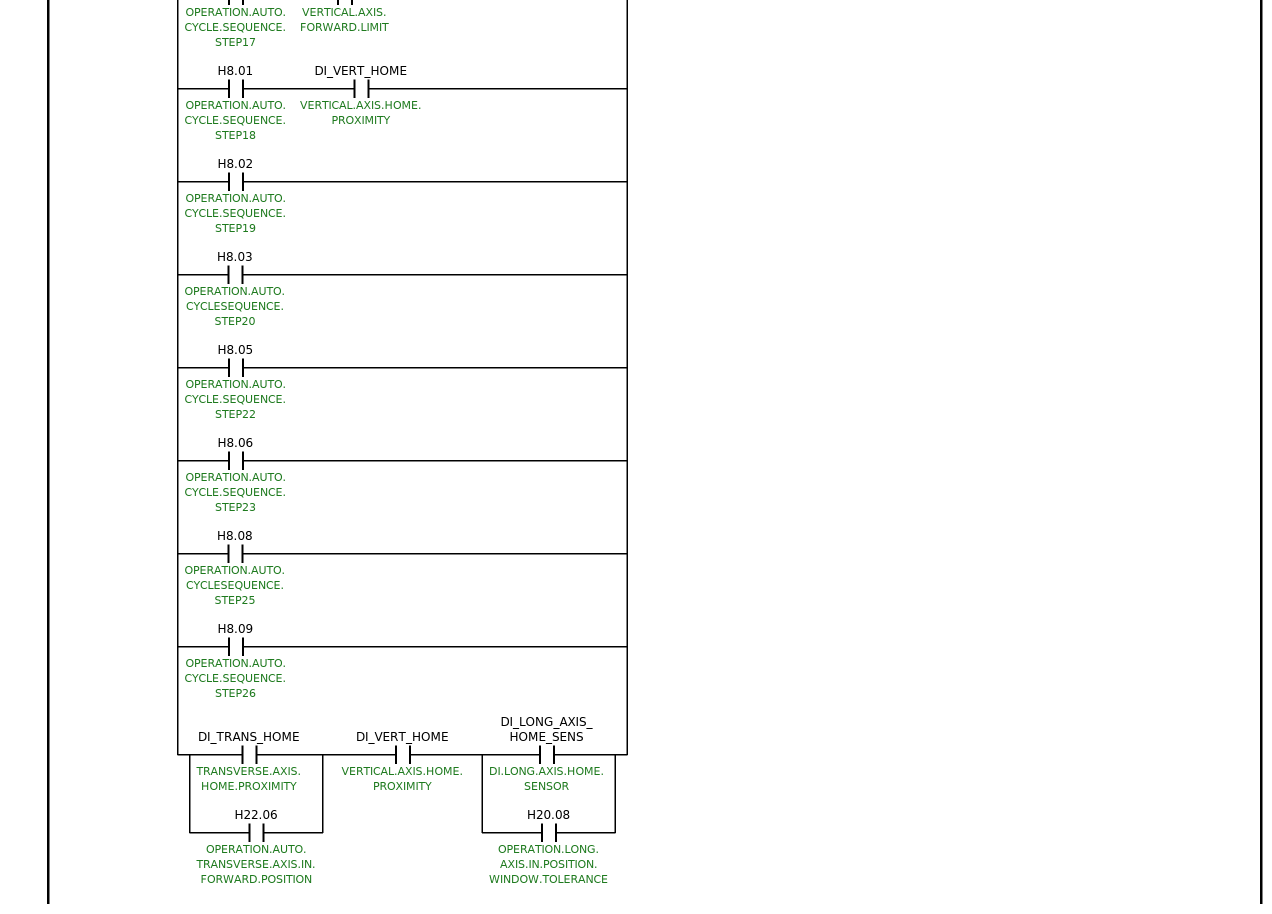
; rung 2
LDNOT H3.02  ; CYCLE.RUN.ACTIVE
LD H7.00  ; OPERATION.AUTO.CYCLE.SEQUENCE.STEP1
OR H7.02  ; OPERATION.AUTO.CYCLE.SEQUENCE.STEP3
OR H7.03  ; OPERATION.AUTO.CYCLE.SEQUENCE.STEP4
OR H7.04  ; OPERATION.AUTO.CYCLE.SEQUENCE.STEP5
LD H7.05  ; OPERATION.AUTO.CYCLE.SEQUENCE.STEP6
AND H22.06  ; OPERATION.AUTO.TRANSVERSE.AXIS.IN.FORWARD.POSITION
ORLD
LD H7.06  ; OPERATION.AUTO.CYCLE.SEQUENCE.STEP7
AND H22.06  ; OPERATION.AUTO.TRANSVERSE.AXIS.IN.FORWARD.POSITION
ORLD
OR H7.07  ; OPERATION.AUTO.CYCLE.SEQUENCE.STEP8
LD H7.08  ; OPERATION.AUTO.CYCLE.SEQUENCE.STEP9
AND H20.08  ; OPERATION.LONG.AXIS.IN.POSITION.WINDOW.TOLERANCE
ORLD
LD H7.09  ; OPERATION.AUTO.CYCLE.SEQUENCE.STEP10
AND H21.08  ; OP.CONTROL.VERTICAL.IN.POSITION
ORLD
OR H7.10  ; OPERATION.AUTO.CYCLE.SEQUENCE.STEP11
LD H7.11  ; OPERATION.AUTO.CYCLE.SEQUENCE.STEP12
AND H21.08  ; OP.CONTROL.VERTICAL.IN.POSITION
ORLD
LD H7.12  ; OPERATION.AUTO.CYCLE.SEQUENCE.STEP13
AND DI_TRANS_HOME  ; TRANSVERSE.AXIS.HOME.PROXIMITY
ORLD
LD H7.13  ; OPERATION.AUTO.CYCLE.SEQUENCE.STEP14
AND H22.06  ; OPERATION.AUTO.TRANSVERSE.AXIS.IN.FORWARD.POSITION
ORLD
LD H7.15  ; OPERATION.AUTO.CYCLE.SEQUENCE.STEP16
AND DI_TRANS_HOME  ; TRANSVERSE.AXIS.HOME.PROXIMITY
ORLD
LD H8.00  ; OPERATION.AUTO.CYCLE.SEQUENCE.STEP17
AND DI_VERT_FWD  ; VERTICAL.AXIS.FORWARD.LIMIT
ORLD
LD H8.01  ; OPERATION.AUTO.CYCLE.SEQUENCE.STEP18
AND DI_VERT_HOME  ; VERTICAL.AXIS.HOME.PROXIMITY
ORLD
OR H8.02  ; OPERATION.AUTO.CYCLE.SEQUENCE.STEP19
OR H8.03  ; OPERATION.AUTO.CYCLESEQUENCE.STEP20
OR H8.05  ; OPERATION.AUTO.CYCLE.SEQUENCE.STEP22
OR H8.06  ; OPERATION.AUTO.CYCLE.SEQUENCE.STEP23
OR H8.08  ; OPERATION.AUTO.CYCLESEQUENCE.STEP25
OR H8.09  ; OPERATION.AUTO.CYCLE.SEQUENCE.STEP26
LD DI_TRANS_HOME  ; TRANSVERSE.AXIS.HOME.PROXIMITY
OR H22.06  ; OPERATION.AUTO.TRANSVERSE.AXIS.IN.FORWARD.POSITION
AND DI_VERT_HOME  ; VERTICAL.AXIS.HOME.PROXIMITY
LD DI_LONG_AXIS_HOME_SENS  ; DI.LONG.AXIS.HOME.SENSOR
OR H20.08  ; OPERATION.LONG.AXIS.IN.POSITION.WINDOW.TOLERANCE
ANDLD
ORLD
ANDLD
AND OI_CTRL_CYCLE_START  ; OI.CONTROL.AUTOMATIC.CYCLE.START.PB
ANDNOT H3.15  ; Cycle Completed
ANDNOT H3.03  ; MACHINE.CYCLE.STOP
AND SAFETY_GATE_OK  ; SAFETY.GATE.OKAY
OUT H2.05  ; OPERATION.AUTO.CYCLE.START.COMMAND

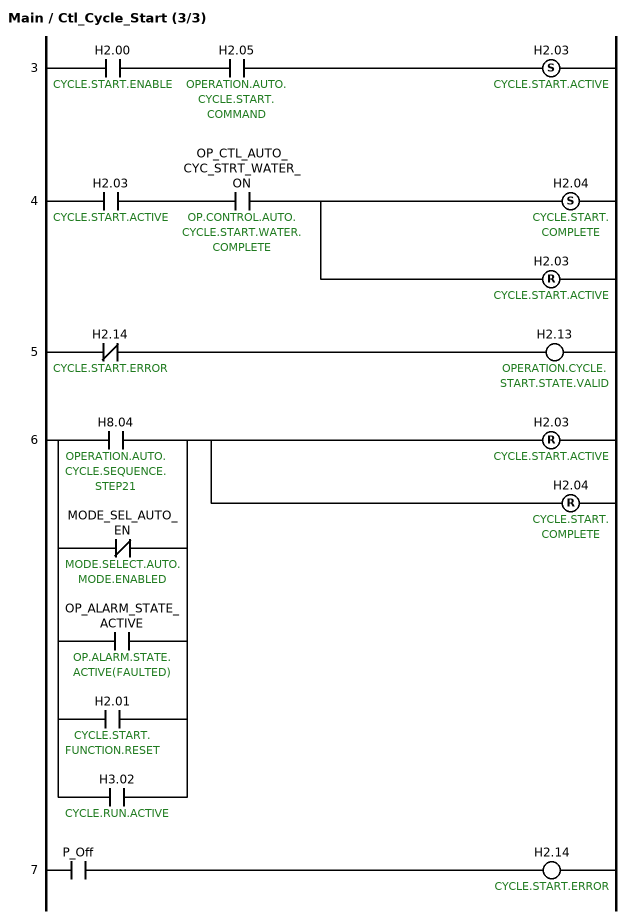
; rung 3
LD H2.00  ; CYCLE.START.ENABLE
AND H2.05  ; OPERATION.AUTO.CYCLE.START.COMMAND
SET H2.03  ; CYCLE.START.ACTIVE
; rung 4
LD H2.03  ; CYCLE.START.ACTIVE
AND OP_CTL_AUTO_CYC_STRT_WATER_ON  ; OP.CONTROL.AUTO.CYCLE.START.WATER.COMPLETE
SET H2.04  ; CYCLE.START.COMPLETE
RSET H2.03  ; CYCLE.START.ACTIVE
; rung 5
LDNOT H2.14  ; CYCLE.START.ERROR
OUT H2.13  ; OPERATION.CYCLE.START.STATE.VALID
; rung 6
LD H8.04  ; OPERATION.AUTO.CYCLE.SEQUENCE.STEP21
ORNOT MODE_SEL_AUTO_EN  ; MODE.SELECT.AUTO.MODE.ENABLED
OR OP_ALARM_STATE_ACTIVE  ; OP.ALARM.STATE.ACTIVE(FAULTED)
OR H2.01  ; CYCLE.START.FUNCTION.RESET
OR H3.02  ; CYCLE.RUN.ACTIVE
RSET H2.03  ; CYCLE.START.ACTIVE
RSET H2.04  ; CYCLE.START.COMPLETE
; rung 7
LD P_Off
OUT H2.14  ; CYCLE.START.ERROR

### Section Ctl_Cycle_Run

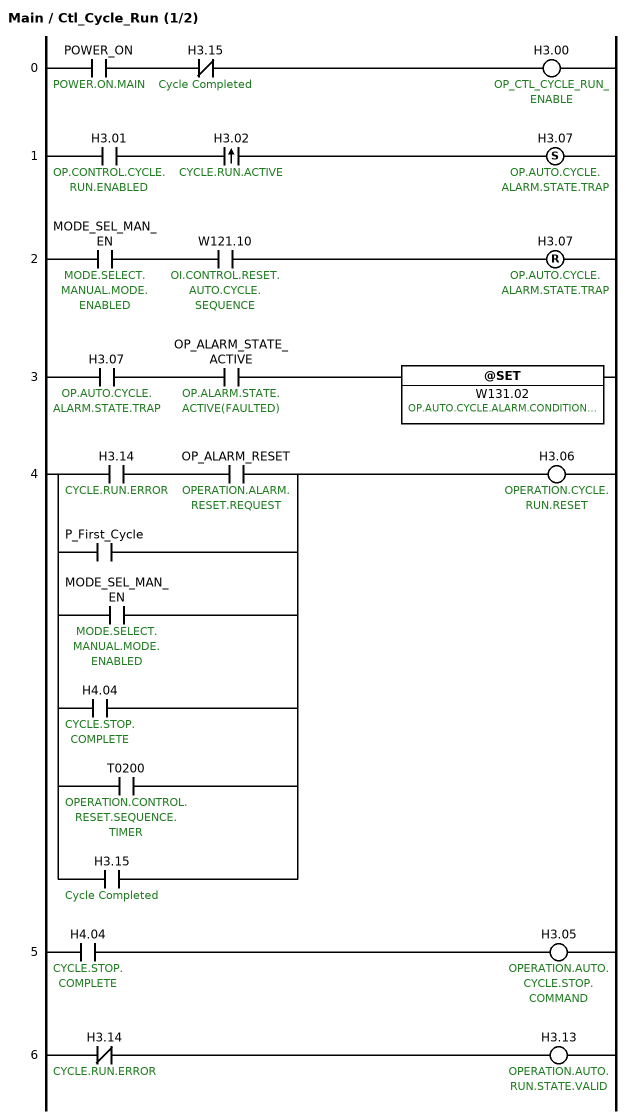
; rung 0
LD POWER_ON  ; POWER.ON.MAIN
ANDNOT H3.15  ; Cycle Completed
OUT H3.00  ; OP_CTL_CYCLE_RUN_ENABLE
; rung 1
LD H3.01  ; OP.CONTROL.CYCLE.RUN.ENABLED
@AND H3.02  ; CYCLE.RUN.ACTIVE
SET H3.07  ; OP.AUTO.CYCLE.ALARM.STATE.TRAP
; rung 2
LD MODE_SEL_MAN_EN  ; MODE.SELECT.MANUAL.MODE.ENABLED
AND W121.10  ; OI.CONTROL.RESET.AUTO.CYCLE.SEQUENCE
RSET H3.07  ; OP.AUTO.CYCLE.ALARM.STATE.TRAP
; rung 3
LD H3.07  ; OP.AUTO.CYCLE.ALARM.STATE.TRAP
AND OP_ALARM_STATE_ACTIVE  ; OP.ALARM.STATE.ACTIVE(FAULTED)
@SET W131.02  ; OP.AUTO.CYCLE.ALARM.CONDITION.IN.CYCLE.MESSAGE.SHOW
; rung 4
LD H3.14  ; CYCLE.RUN.ERROR
AND OP_ALARM_RESET  ; OPERATION.ALARM.RESET.REQUEST
OR P_First_Cycle
OR MODE_SEL_MAN_EN  ; MODE.SELECT.MANUAL.MODE.ENABLED
OR H4.04  ; CYCLE.STOP.COMPLETE
OR T0200  ; OPERATION.CONTROL.RESET.SEQUENCE.TIMER
OR H3.15  ; Cycle Completed
OUT H3.06  ; OPERATION.CYCLE.RUN.RESET
; rung 5
LD H4.04  ; CYCLE.STOP.COMPLETE
OUT H3.05  ; OPERATION.AUTO.CYCLE.STOP.COMMAND
; rung 6
LDNOT H3.14  ; CYCLE.RUN.ERROR
OUT H3.13  ; OPERATION.AUTO.RUN.STATE.VALID

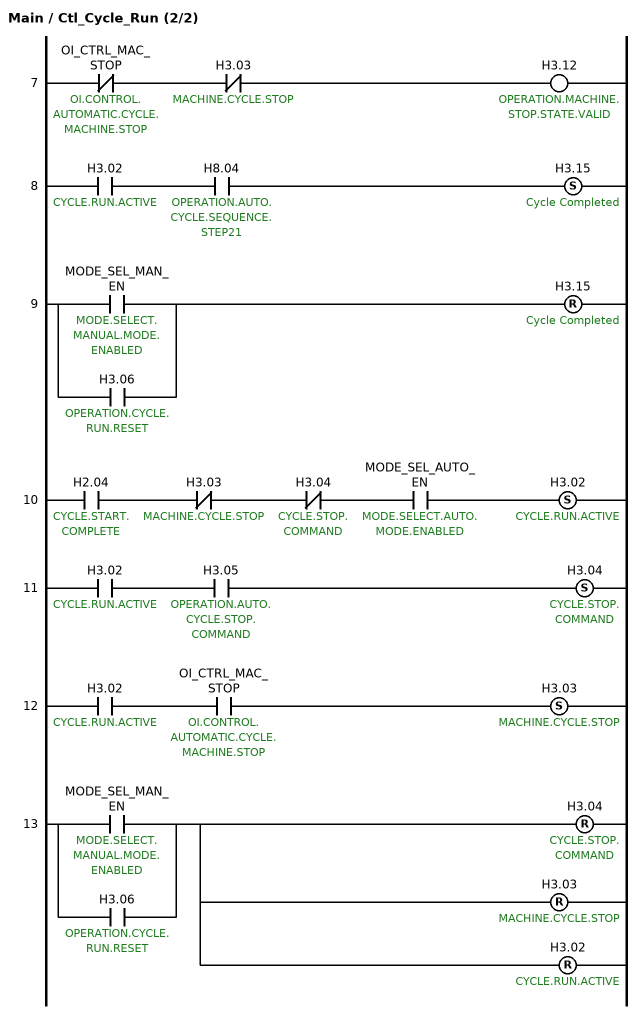
; rung 7
LDNOT OI_CTRL_MAC_STOP  ; OI.CONTROL.AUTOMATIC.CYCLE.MACHINE.STOP
ANDNOT H3.03  ; MACHINE.CYCLE.STOP
OUT H3.12  ; OPERATION.MACHINE.STOP.STATE.VALID
; rung 8
LD H3.02  ; CYCLE.RUN.ACTIVE
AND H8.04  ; OPERATION.AUTO.CYCLE.SEQUENCE.STEP21
SET H3.15  ; Cycle Completed
; rung 9
LD MODE_SEL_MAN_EN  ; MODE.SELECT.MANUAL.MODE.ENABLED
OR H3.06  ; OPERATION.CYCLE.RUN.RESET
RSET H3.15  ; Cycle Completed
; rung 10
LD H2.04  ; CYCLE.START.COMPLETE
ANDNOT H3.03  ; MACHINE.CYCLE.STOP
ANDNOT H3.04  ; CYCLE.STOP.COMMAND
AND MODE_SEL_AUTO_EN  ; MODE.SELECT.AUTO.MODE.ENABLED
SET H3.02  ; CYCLE.RUN.ACTIVE
; rung 11
LD H3.02  ; CYCLE.RUN.ACTIVE
AND H3.05  ; OPERATION.AUTO.CYCLE.STOP.COMMAND
SET H3.04  ; CYCLE.STOP.COMMAND
; rung 12
LD H3.02  ; CYCLE.RUN.ACTIVE
AND OI_CTRL_MAC_STOP  ; OI.CONTROL.AUTOMATIC.CYCLE.MACHINE.STOP
SET H3.03  ; MACHINE.CYCLE.STOP
; rung 13
LD MODE_SEL_MAN_EN  ; MODE.SELECT.MANUAL.MODE.ENABLED
OR H3.06  ; OPERATION.CYCLE.RUN.RESET
RSET H3.04  ; CYCLE.STOP.COMMAND
RSET H3.03  ; MACHINE.CYCLE.STOP
RSET H3.02  ; CYCLE.RUN.ACTIVE

### Section Ctl_Cycle_Stop

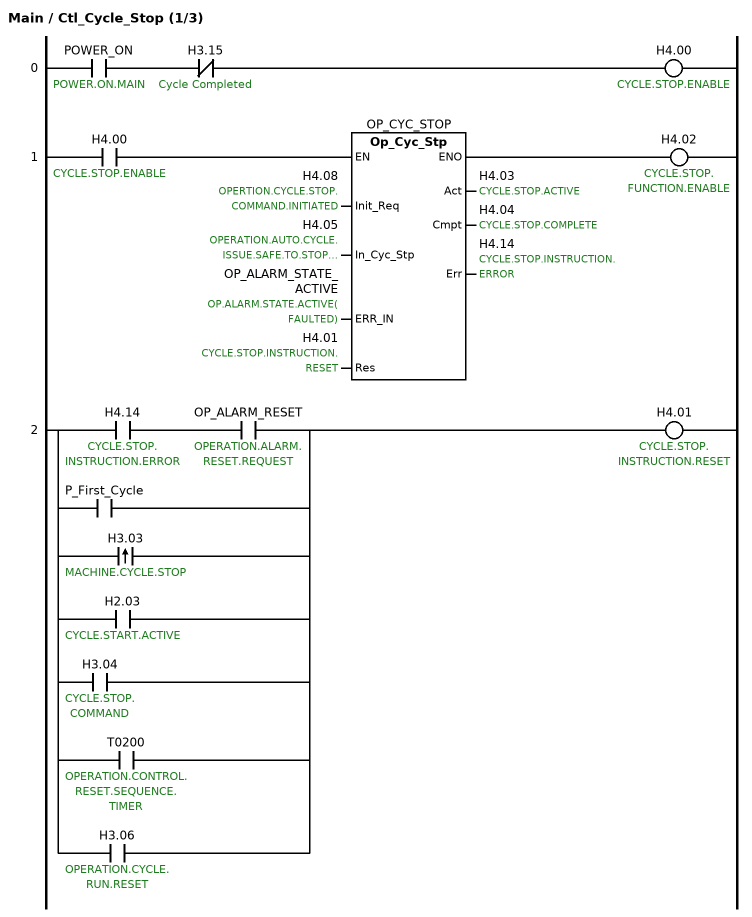
; rung 0
LD POWER_ON  ; POWER.ON.MAIN
ANDNOT H3.15  ; Cycle Completed
OUT H4.00  ; CYCLE.STOP.ENABLE
; rung 1
LD H4.00  ; CYCLE.STOP.ENABLE
CALL OP_CYC_STOP : Op_Cyc_Stp (Init_Req := H4.08, In_Cyc_Stp := H4.05, ERR_IN := OP_ALARM_STATE_ACTIVE, Res := H4.01, Act => H4.03, Cmpt => H4.04, Err => H4.14)  ; OPERTION.CYCLE.STOP.COMMAND.INITIATED, OPERATION.AUTO.CYCLE.ISSUE.SAFE.TO.STOP.COMMAND, OP.ALARM.STATE.ACTIVE(FAULTED), CYCLE.STOP.INSTRUCTION.RESET, CYCLE.STOP.ACTIVE, CYCLE.STOP.COMPLETE, CYCLE.STOP.INSTRUCTION.ERROR
OUT H4.02  ; CYCLE.STOP.FUNCTION.ENABLE
; rung 2
LD H4.14  ; CYCLE.STOP.INSTRUCTION.ERROR
AND OP_ALARM_RESET  ; OPERATION.ALARM.RESET.REQUEST
OR P_First_Cycle
@OR H3.03  ; MACHINE.CYCLE.STOP
OR H2.03  ; CYCLE.START.ACTIVE
OR H3.04  ; CYCLE.STOP.COMMAND
OR T0200  ; OPERATION.CONTROL.RESET.SEQUENCE.TIMER
OR H3.06  ; OPERATION.CYCLE.RUN.RESET
OUT H4.01  ; CYCLE.STOP.INSTRUCTION.RESET

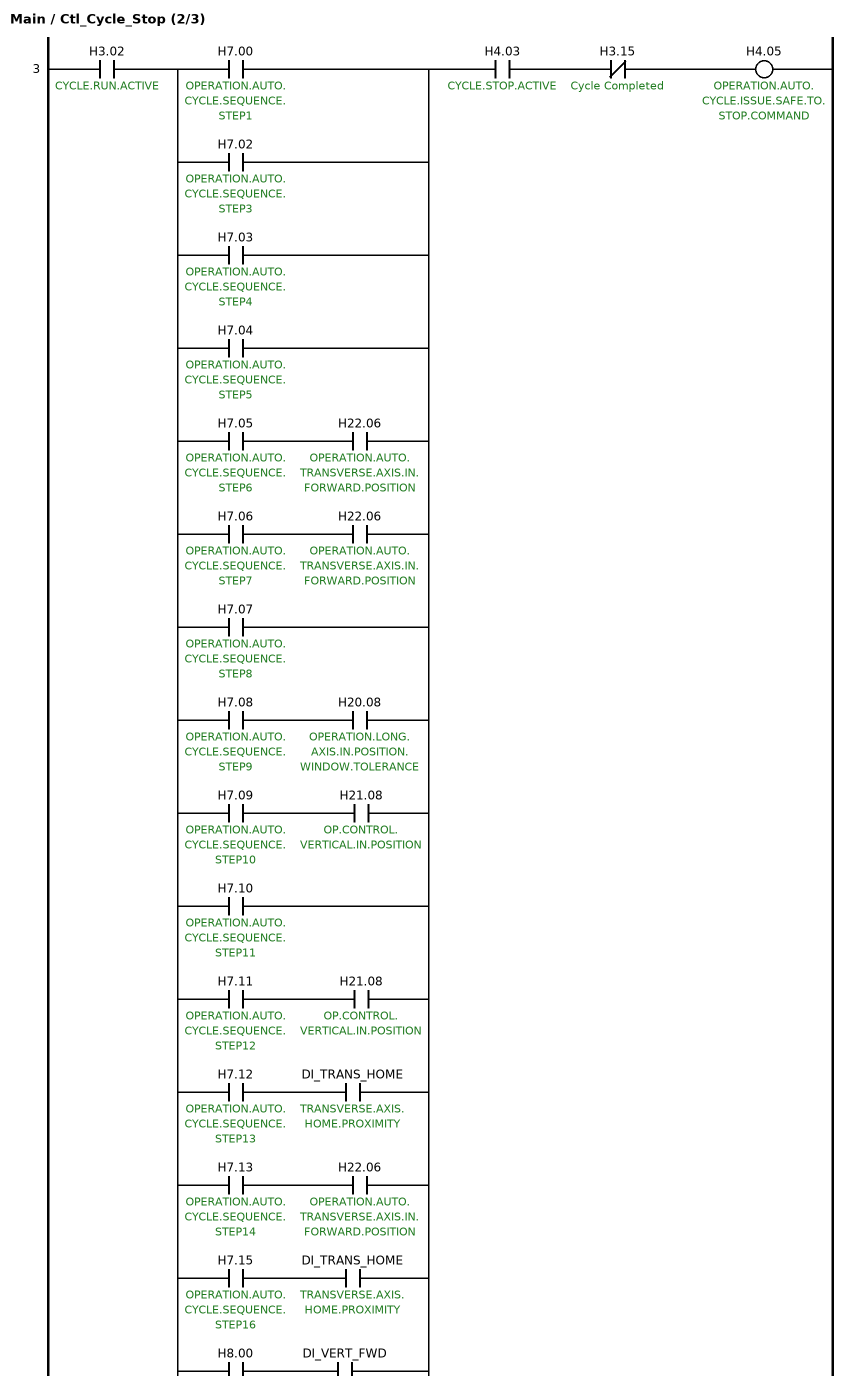

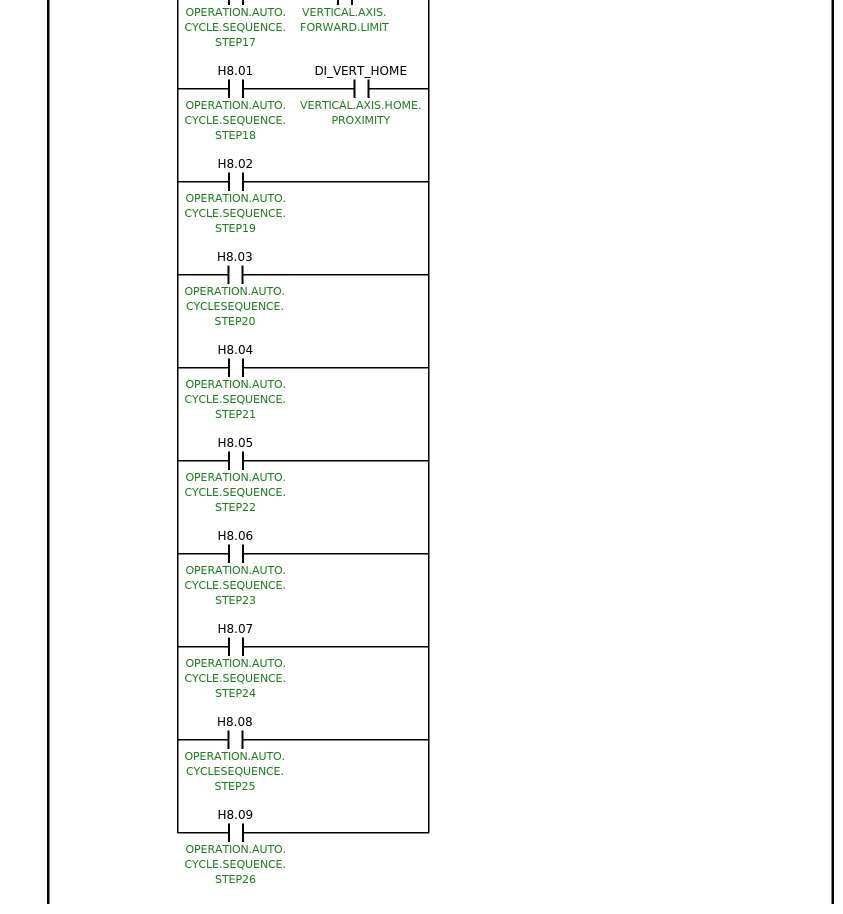
; rung 3
LD H3.02  ; CYCLE.RUN.ACTIVE
LD H7.00  ; OPERATION.AUTO.CYCLE.SEQUENCE.STEP1
OR H7.02  ; OPERATION.AUTO.CYCLE.SEQUENCE.STEP3
OR H7.03  ; OPERATION.AUTO.CYCLE.SEQUENCE.STEP4
OR H7.04  ; OPERATION.AUTO.CYCLE.SEQUENCE.STEP5
LD H7.05  ; OPERATION.AUTO.CYCLE.SEQUENCE.STEP6
AND H22.06  ; OPERATION.AUTO.TRANSVERSE.AXIS.IN.FORWARD.POSITION
ORLD
LD H7.06  ; OPERATION.AUTO.CYCLE.SEQUENCE.STEP7
AND H22.06  ; OPERATION.AUTO.TRANSVERSE.AXIS.IN.FORWARD.POSITION
ORLD
OR H7.07  ; OPERATION.AUTO.CYCLE.SEQUENCE.STEP8
LD H7.08  ; OPERATION.AUTO.CYCLE.SEQUENCE.STEP9
AND H20.08  ; OPERATION.LONG.AXIS.IN.POSITION.WINDOW.TOLERANCE
ORLD
LD H7.09  ; OPERATION.AUTO.CYCLE.SEQUENCE.STEP10
AND H21.08  ; OP.CONTROL.VERTICAL.IN.POSITION
ORLD
OR H7.10  ; OPERATION.AUTO.CYCLE.SEQUENCE.STEP11
LD H7.11  ; OPERATION.AUTO.CYCLE.SEQUENCE.STEP12
AND H21.08  ; OP.CONTROL.VERTICAL.IN.POSITION
ORLD
LD H7.12  ; OPERATION.AUTO.CYCLE.SEQUENCE.STEP13
AND DI_TRANS_HOME  ; TRANSVERSE.AXIS.HOME.PROXIMITY
ORLD
LD H7.13  ; OPERATION.AUTO.CYCLE.SEQUENCE.STEP14
AND H22.06  ; OPERATION.AUTO.TRANSVERSE.AXIS.IN.FORWARD.POSITION
ORLD
LD H7.15  ; OPERATION.AUTO.CYCLE.SEQUENCE.STEP16
AND DI_TRANS_HOME  ; TRANSVERSE.AXIS.HOME.PROXIMITY
ORLD
LD H8.00  ; OPERATION.AUTO.CYCLE.SEQUENCE.STEP17
AND DI_VERT_FWD  ; VERTICAL.AXIS.FORWARD.LIMIT
ORLD
LD H8.01  ; OPERATION.AUTO.CYCLE.SEQUENCE.STEP18
AND DI_VERT_HOME  ; VERTICAL.AXIS.HOME.PROXIMITY
ORLD
OR H8.02  ; OPERATION.AUTO.CYCLE.SEQUENCE.STEP19
OR H8.03  ; OPERATION.AUTO.CYCLESEQUENCE.STEP20
OR H8.04  ; OPERATION.AUTO.CYCLE.SEQUENCE.STEP21
OR H8.05  ; OPERATION.AUTO.CYCLE.SEQUENCE.STEP22
OR H8.06  ; OPERATION.AUTO.CYCLE.SEQUENCE.STEP23
OR H8.07  ; OPERATION.AUTO.CYCLE.SEQUENCE.STEP24
OR H8.08  ; OPERATION.AUTO.CYCLESEQUENCE.STEP25
OR H8.09  ; OPERATION.AUTO.CYCLE.SEQUENCE.STEP26
ANDLD
AND H4.03  ; CYCLE.STOP.ACTIVE
ANDNOT H3.15  ; Cycle Completed
OUT H4.05  ; OPERATION.AUTO.CYCLE.ISSUE.SAFE.TO.STOP.COMMAND

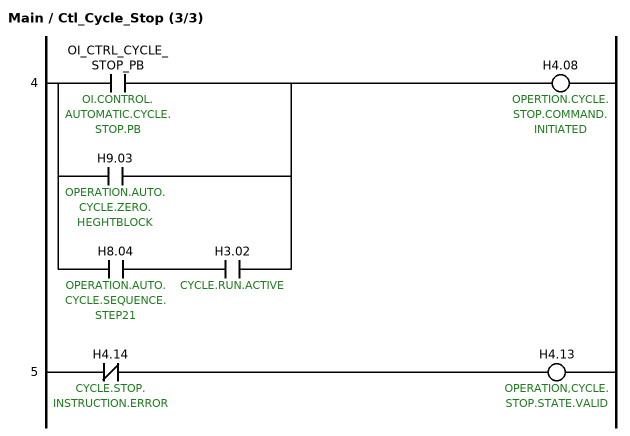
; rung 4
LD OI_CTRL_CYCLE_STOP_PB  ; OI.CONTROL.AUTOMATIC.CYCLE.STOP.PB
OR H9.03  ; OPERATION.AUTO.CYCLE.ZERO.HEGHTBLOCK
LD H8.04  ; OPERATION.AUTO.CYCLE.SEQUENCE.STEP21
AND H3.02  ; CYCLE.RUN.ACTIVE
ORLD
OUT H4.08  ; OPERTION.CYCLE.STOP.COMMAND.INITIATED
; rung 5
LDNOT H4.14  ; CYCLE.STOP.INSTRUCTION.ERROR
OUT H4.13  ; OPERATION,CYCLE.STOP.STATE.VALID

### Section Ctl_Auto_Cycle_Sequence

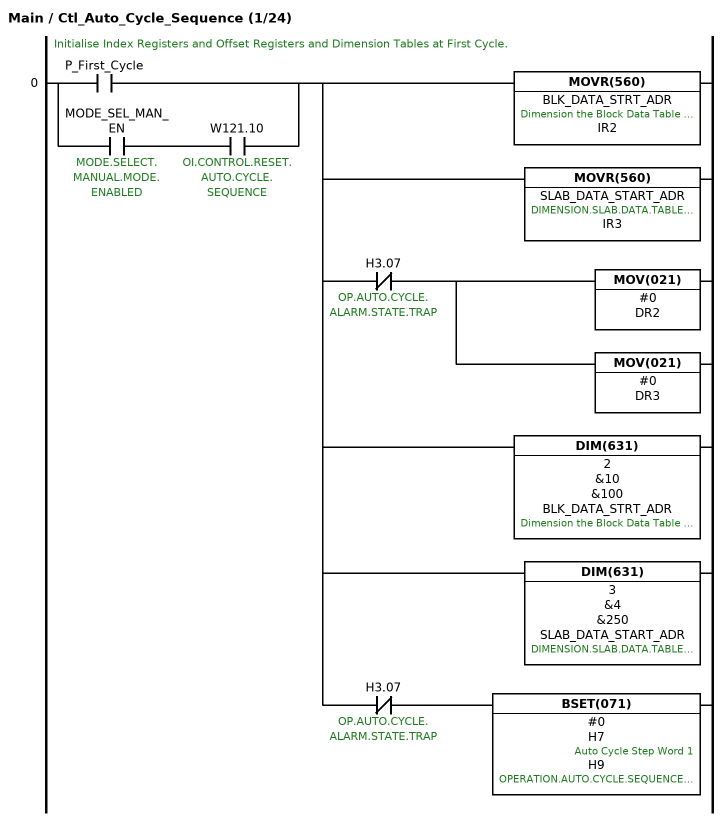
; rung 0: Initialise Index Registers and Offset Registers and Dimension Tables at First Cycle.
LD P_First_Cycle
LD MODE_SEL_MAN_EN  ; MODE.SELECT.MANUAL.MODE.ENABLED
AND W121.10  ; OI.CONTROL.RESET.AUTO.CYCLE.SEQUENCE
ORLD
OUT TR0
MOVR(560) BLK_DATA_STRT_ADR IR2  ; Dimension the Block Data Table - Start Address
MOVR(560) SLAB_DATA_START_ADR IR3  ; DIMENSION.SLAB.DATA.TABLE.START.ADDRESS
ANDNOT H3.07  ; OP.AUTO.CYCLE.ALARM.STATE.TRAP
MOV(021) #0 DR2
MOV(021) #0 DR3
LD TR0
DIM(631) 2 &10 &100 BLK_DATA_STRT_ADR  ; Dimension the Block Data Table - Start Address
DIM(631) 3 &4 &250 SLAB_DATA_START_ADR  ; DIMENSION.SLAB.DATA.TABLE.START.ADDRESS
ANDNOT H3.07  ; OP.AUTO.CYCLE.ALARM.STATE.TRAP
BSET(071) #0 H7 H9  ; Auto Cycle Step Word 1, OPERATION.AUTO.CYCLE.SEQUENCE.STATE.BITS

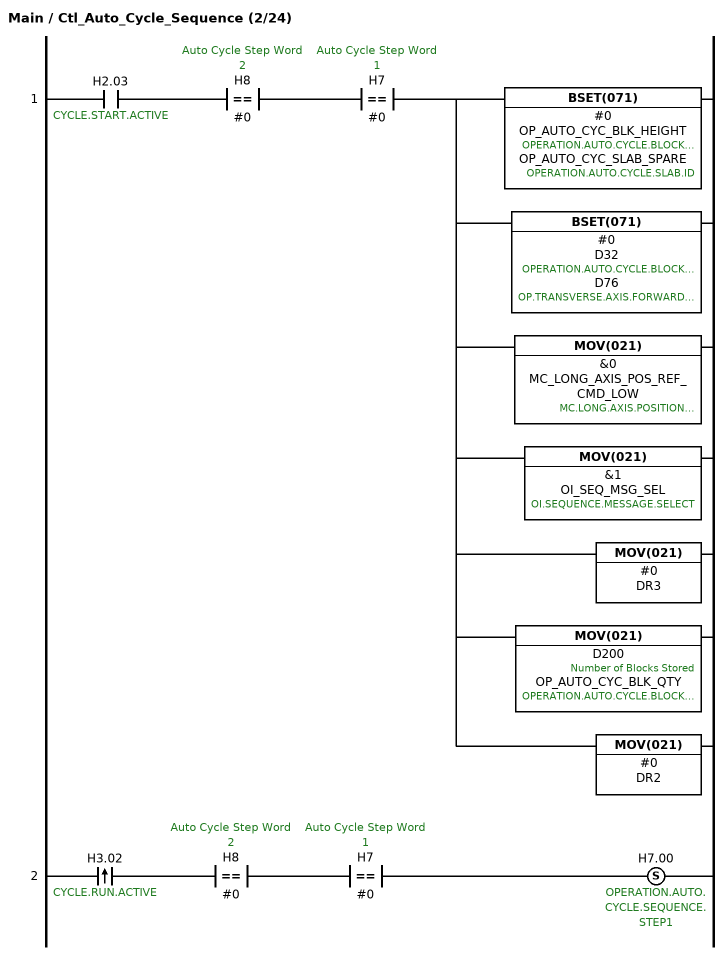
; rung 1
LD H2.03  ; CYCLE.START.ACTIVE
AND=(300) H8 #0  ; Auto Cycle Step Word 2
AND=(300) H7 #0  ; Auto Cycle Step Word 1
BSET(071) #0 OP_AUTO_CYC_BLK_HEIGHT OP_AUTO_CYC_SLAB_SPARE  ; OPERATION.AUTO.CYCLE.BLOCK.HEIGHT.WORKING, OPERATION.AUTO.CYCLE.SLAB.ID
BSET(071) #0 D32 D76  ; OPERATION.AUTO.CYCLE.BLOCK.FIRST.CUT.WORKING.REAL, OP.TRANSVERSE.AXIS.FORWARD.TARGET
MOV(021) &0 MC_LONG_AXIS_POS_REF_CMD_LOW  ; MC.LONG.AXIS.POSITION.REFERENCE.COMMAND.VALUE.LOW.WORD
MOV(021) &1 OI_SEQ_MSG_SEL  ; OI.SEQUENCE.MESSAGE.SELECT
MOV(021) #0 DR3
MOV(021) D200 OP_AUTO_CYC_BLK_QTY  ; Number of Blocks Stored, OPERATION.AUTO.CYCLE.BLOCK.QUANTITY
MOV(021) #0 DR2
; rung 2
@LD H3.02  ; CYCLE.RUN.ACTIVE
AND=(300) H8 #0  ; Auto Cycle Step Word 2
AND=(300) H7 #0  ; Auto Cycle Step Word 1
SET H7.00  ; OPERATION.AUTO.CYCLE.SEQUENCE.STEP1

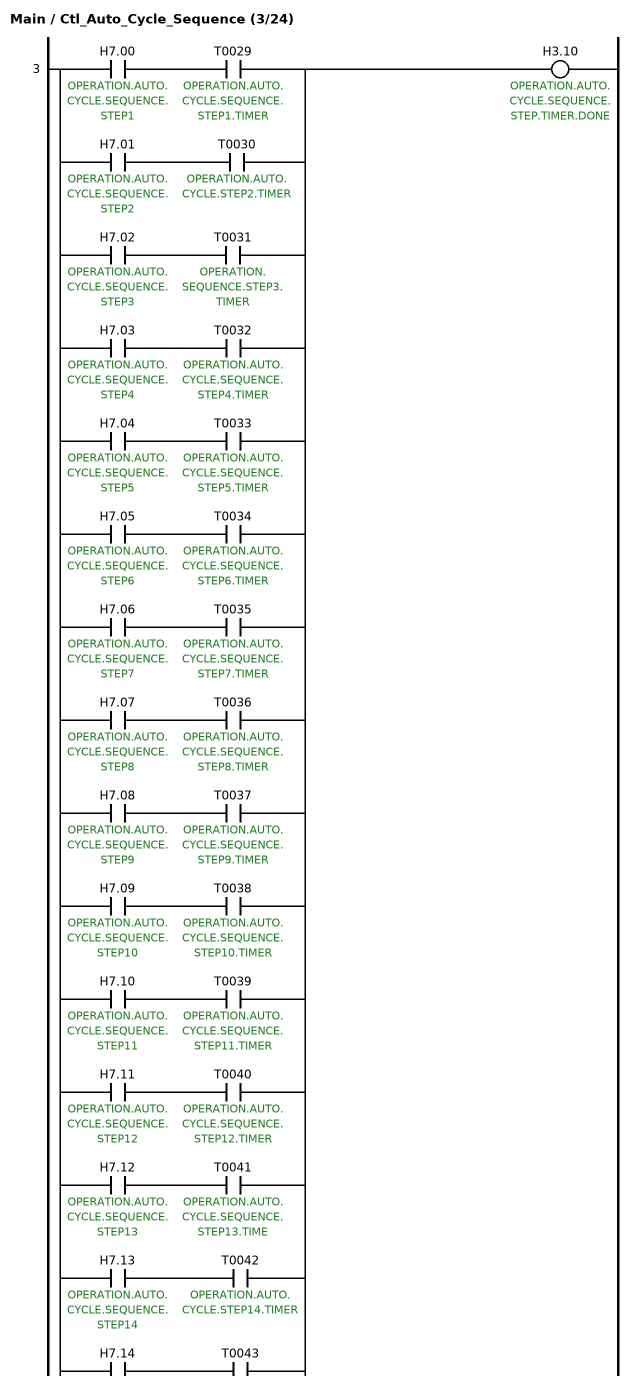

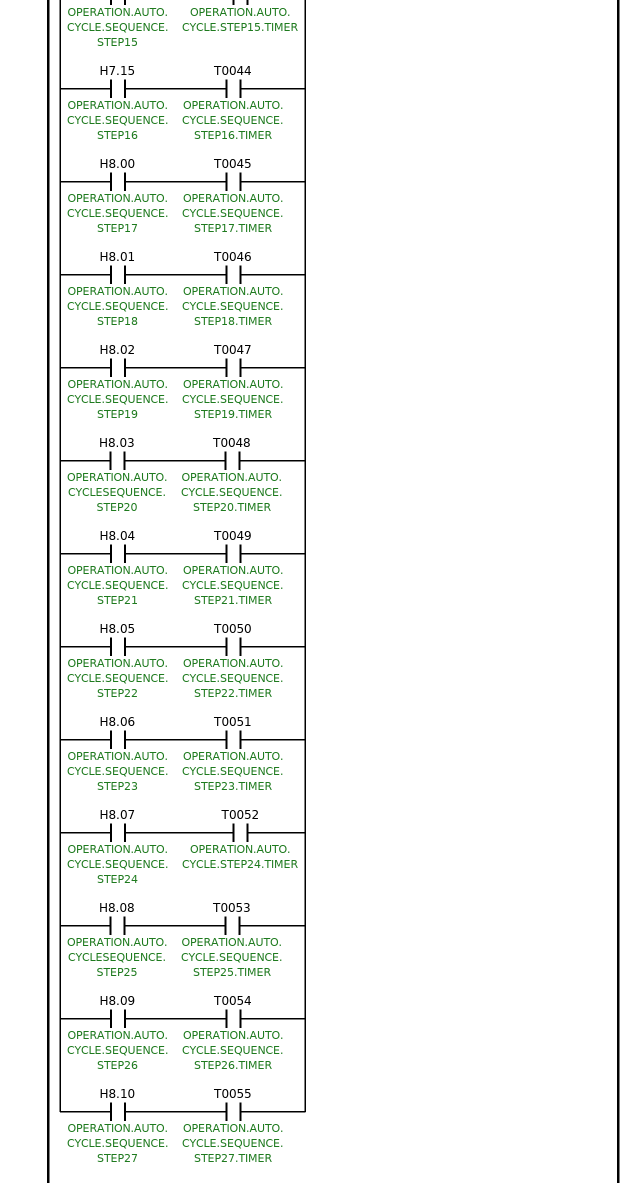
; rung 3
LD H7.00  ; OPERATION.AUTO.CYCLE.SEQUENCE.STEP1
AND T0029  ; OPERATION.AUTO.CYCLE.SEQUENCE.STEP1.TIMER
LD H7.01  ; OPERATION.AUTO.CYCLE.SEQUENCE.STEP2
AND T0030  ; OPERATION.AUTO.CYCLE.STEP2.TIMER
ORLD
LD H7.02  ; OPERATION.AUTO.CYCLE.SEQUENCE.STEP3
AND T0031  ; OPERATION.SEQUENCE.STEP3.TIMER
ORLD
LD H7.03  ; OPERATION.AUTO.CYCLE.SEQUENCE.STEP4
AND T0032  ; OPERATION.AUTO.CYCLE.SEQUENCE.STEP4.TIMER
ORLD
LD H7.04  ; OPERATION.AUTO.CYCLE.SEQUENCE.STEP5
AND T0033  ; OPERATION.AUTO.CYCLE.SEQUENCE.STEP5.TIMER
ORLD
LD H7.05  ; OPERATION.AUTO.CYCLE.SEQUENCE.STEP6
AND T0034  ; OPERATION.AUTO.CYCLE.SEQUENCE.STEP6.TIMER
ORLD
LD H7.06  ; OPERATION.AUTO.CYCLE.SEQUENCE.STEP7
AND T0035  ; OPERATION.AUTO.CYCLE.SEQUENCE.STEP7.TIMER
ORLD
LD H7.07  ; OPERATION.AUTO.CYCLE.SEQUENCE.STEP8
AND T0036  ; OPERATION.AUTO.CYCLE.SEQUENCE.STEP8.TIMER
ORLD
LD H7.08  ; OPERATION.AUTO.CYCLE.SEQUENCE.STEP9
AND T0037  ; OPERATION.AUTO.CYCLE.SEQUENCE.STEP9.TIMER
ORLD
LD H7.09  ; OPERATION.AUTO.CYCLE.SEQUENCE.STEP10
AND T0038  ; OPERATION.AUTO.CYCLE.SEQUENCE.STEP10.TIMER
ORLD
LD H7.10  ; OPERATION.AUTO.CYCLE.SEQUENCE.STEP11
AND T0039  ; OPERATION.AUTO.CYCLE.SEQUENCE.STEP11.TIMER
ORLD
LD H7.11  ; OPERATION.AUTO.CYCLE.SEQUENCE.STEP12
AND T0040  ; OPERATION.AUTO.CYCLE.SEQUENCE.STEP12.TIMER
ORLD
LD H7.12  ; OPERATION.AUTO.CYCLE.SEQUENCE.STEP13
AND T0041  ; OPERATION.AUTO.CYCLE.SEQUENCE.STEP13.TIME
ORLD
LD H7.13  ; OPERATION.AUTO.CYCLE.SEQUENCE.STEP14
AND T0042  ; OPERATION.AUTO.CYCLE.STEP14.TIMER
ORLD
LD H7.14  ; OPERATION.AUTO.CYCLE.SEQUENCE.STEP15
AND T0043  ; OPERATION.AUTO.CYCLE.STEP15.TIMER
ORLD
LD H7.15  ; OPERATION.AUTO.CYCLE.SEQUENCE.STEP16
AND T0044  ; OPERATION.AUTO.CYCLE.SEQUENCE.STEP16.TIMER
ORLD
LD H8.00  ; OPERATION.AUTO.CYCLE.SEQUENCE.STEP17
AND T0045  ; OPERATION.AUTO.CYCLE.SEQUENCE.STEP17.TIMER
ORLD
LD H8.01  ; OPERATION.AUTO.CYCLE.SEQUENCE.STEP18
AND T0046  ; OPERATION.AUTO.CYCLE.SEQUENCE.STEP18.TIMER
ORLD
LD H8.02  ; OPERATION.AUTO.CYCLE.SEQUENCE.STEP19
AND T0047  ; OPERATION.AUTO.CYCLE.SEQUENCE.STEP19.TIMER
ORLD
LD H8.03  ; OPERATION.AUTO.CYCLESEQUENCE.STEP20
AND T0048  ; OPERATION.AUTO.CYCLE.SEQUENCE.STEP20.TIMER
ORLD
LD H8.04  ; OPERATION.AUTO.CYCLE.SEQUENCE.STEP21
AND T0049  ; OPERATION.AUTO.CYCLE.SEQUENCE.STEP21.TIMER
ORLD
LD H8.05  ; OPERATION.AUTO.CYCLE.SEQUENCE.STEP22
AND T0050  ; OPERATION.AUTO.CYCLE.SEQUENCE.STEP22.TIMER
ORLD
LD H8.06  ; OPERATION.AUTO.CYCLE.SEQUENCE.STEP23
AND T0051  ; OPERATION.AUTO.CYCLE.SEQUENCE.STEP23.TIMER
ORLD
LD H8.07  ; OPERATION.AUTO.CYCLE.SEQUENCE.STEP24
AND T0052  ; OPERATION.AUTO.CYCLE.STEP24.TIMER
ORLD
LD H8.08  ; OPERATION.AUTO.CYCLESEQUENCE.STEP25
AND T0053  ; OPERATION.AUTO.CYCLE.SEQUENCE.STEP25.TIMER
ORLD
LD H8.09  ; OPERATION.AUTO.CYCLE.SEQUENCE.STEP26
AND T0054  ; OPERATION.AUTO.CYCLE.SEQUENCE.STEP26.TIMER
ORLD
LD H8.10  ; OPERATION.AUTO.CYCLE.SEQUENCE.STEP27
AND T0055  ; OPERATION.AUTO.CYCLE.SEQUENCE.STEP27.TIMER
ORLD
OUT H3.10  ; OPERATION.AUTO.CYCLE.SEQUENCE.STEP.TIMER.DONE

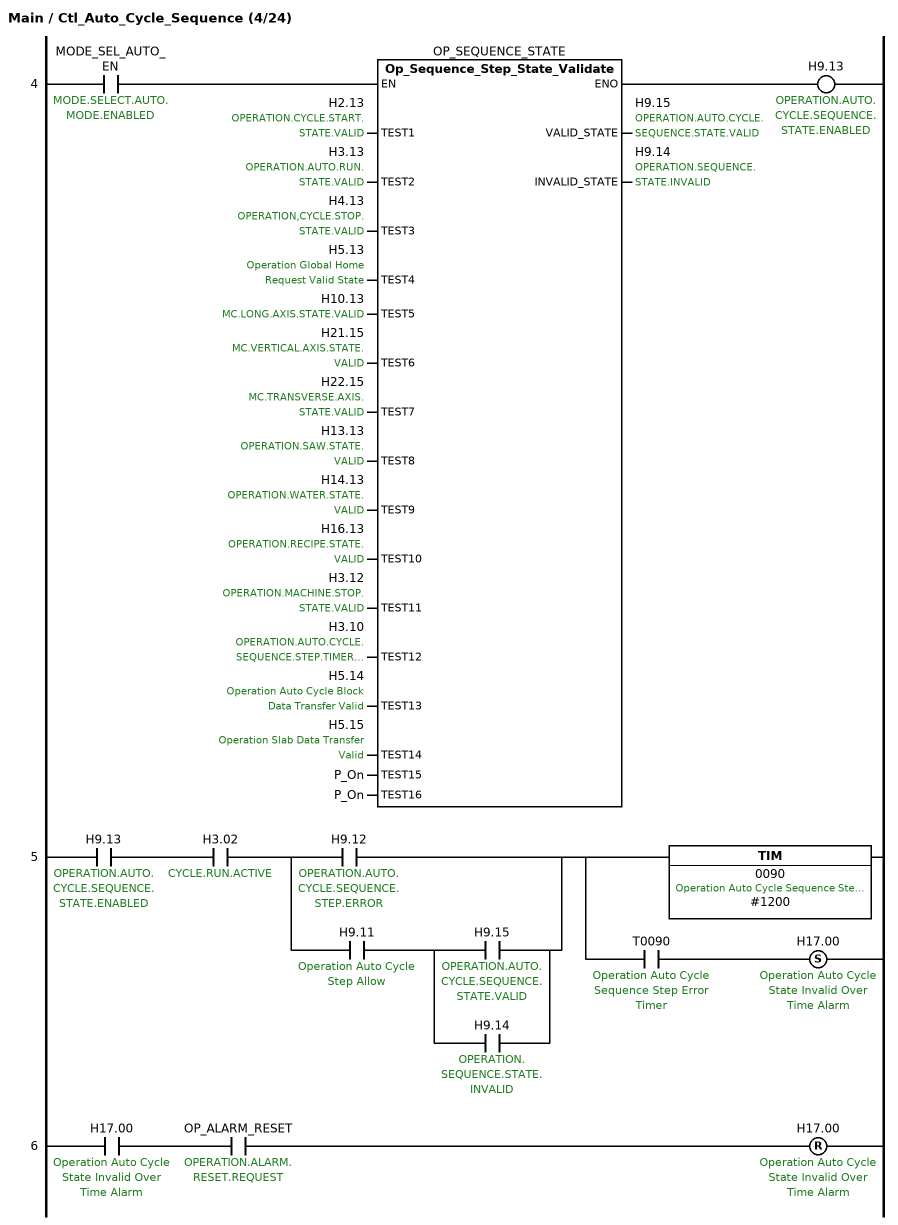
; rung 4
LD MODE_SEL_AUTO_EN  ; MODE.SELECT.AUTO.MODE.ENABLED
CALL OP_SEQUENCE_STATE : Op_Sequence_Step_State_Validate (TEST1 := H2.13, TEST2 := H3.13, TEST3 := H4.13, TEST4 := H5.13, TEST5 := H10.13, TEST6 := H21.15, TEST7 := H22.15, TEST8 := H13.13, TEST9 := H14.13, TEST10 := H16.13, TEST11 := H3.12, TEST12 := H3.10, TEST13 := H5.14, TEST14 := H5.15, TEST15 := P_On, TEST16 := P_On, VALID_STATE => H9.15, INVALID_STATE => H9.14)  ; OPERATION.CYCLE.START.STATE.VALID, OPERATION.AUTO.RUN.STATE.VALID, OPERATION,CYCLE.STOP.STATE.VALID, Operation Global Home Request Valid State, MC.LONG.AXIS.STATE.VALID, MC.VERTICAL.AXIS.STATE.VALID, MC.TRANSVERSE.AXIS.STATE.VALID, OPERATION.SAW.STATE.VALID, OPERATION.WATER.STATE.VALID, OPERATION.RECIPE.STATE.VALID, OPERATION.MACHINE.STOP.STATE.VALID, OPERATION.AUTO.CYCLE.SEQUENCE.STEP.TIMER.DONE, Operation Auto Cycle Block Data Transfer Valid, Operation Slab Data Transfer Valid, OPERATION.AUTO.CYCLE.SEQUENCE.STATE.VALID, OPERATION.SEQUENCE.STATE.INVALID
OUT H9.13  ; OPERATION.AUTO.CYCLE.SEQUENCE.STATE.ENABLED
; rung 5
LD H9.13  ; OPERATION.AUTO.CYCLE.SEQUENCE.STATE.ENABLED
AND H3.02  ; CYCLE.RUN.ACTIVE
LD H9.12  ; OPERATION.AUTO.CYCLE.SEQUENCE.STEP.ERROR
LD H9.11  ; Operation Auto Cycle Step Allow
LD H9.15  ; OPERATION.AUTO.CYCLE.SEQUENCE.STATE.VALID
OR H9.14  ; OPERATION.SEQUENCE.STATE.INVALID
ANDLD
ORLD
ANDLD
TIM 0090 #1200  ; Operation Auto Cycle Sequence Step Error Timer
AND T0090  ; Operation Auto Cycle Sequence Step Error Timer
SET H17.00  ; Operation Auto Cycle State Invalid Over Time Alarm
; rung 6
LD H17.00  ; Operation Auto Cycle State Invalid Over Time Alarm
AND OP_ALARM_RESET  ; OPERATION.ALARM.RESET.REQUEST
RSET H17.00  ; Operation Auto Cycle State Invalid Over Time Alarm

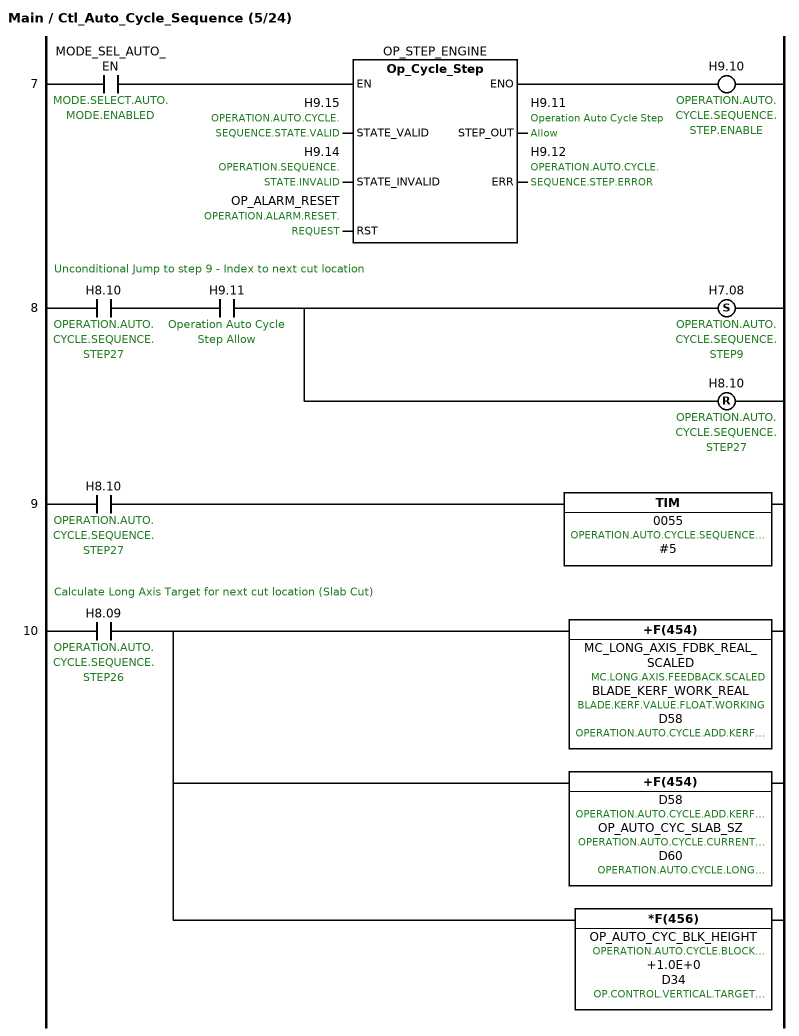
; rung 7
LD MODE_SEL_AUTO_EN  ; MODE.SELECT.AUTO.MODE.ENABLED
CALL OP_STEP_ENGINE : Op_Cycle_Step (STATE_VALID := H9.15, STATE_INVALID := H9.14, RST := OP_ALARM_RESET, STEP_OUT => H9.11, ERR => H9.12)  ; OPERATION.AUTO.CYCLE.SEQUENCE.STATE.VALID, OPERATION.SEQUENCE.STATE.INVALID, OPERATION.ALARM.RESET.REQUEST, Operation Auto Cycle Step Allow, OPERATION.AUTO.CYCLE.SEQUENCE.STEP.ERROR
OUT H9.10  ; OPERATION.AUTO.CYCLE.SEQUENCE.STEP.ENABLE
; rung 8: Unconditional Jump to step 9 - Index to next cut location
LD H8.10  ; OPERATION.AUTO.CYCLE.SEQUENCE.STEP27
AND H9.11  ; Operation Auto Cycle Step Allow
SET H7.08  ; OPERATION.AUTO.CYCLE.SEQUENCE.STEP9
RSET H8.10  ; OPERATION.AUTO.CYCLE.SEQUENCE.STEP27
; rung 9
LD H8.10  ; OPERATION.AUTO.CYCLE.SEQUENCE.STEP27
TIM 0055 #5  ; OPERATION.AUTO.CYCLE.SEQUENCE.STEP27.TIMER
; rung 10: Calculate Long Axis Target for next cut location (Slab Cut)
LD H8.09  ; OPERATION.AUTO.CYCLE.SEQUENCE.STEP26
+F(454) MC_LONG_AXIS_FDBK_REAL_SCALED BLADE_KERF_WORK_REAL D58  ; MC.LONG.AXIS.FEEDBACK.SCALED, BLADE.KERF.VALUE.FLOAT.WORKING, OPERATION.AUTO.CYCLE.ADD.KERF.TO.LOCATION.REAL
+F(454) D58 OP_AUTO_CYC_SLAB_SZ D60  ; OPERATION.AUTO.CYCLE.ADD.KERF.TO.LOCATION.REAL, OPERATION.AUTO.CYCLE.CURRENT.SLAB.SIZE, OPERATION.AUTO.CYCLE.LONG.INDEX.LOCATION.REAL
*F(456) OP_AUTO_CYC_BLK_HEIGHT +1.0E+0 D34  ; OPERATION.AUTO.CYCLE.BLOCK.HEIGHT.WORKING, OP.CONTROL.VERTICAL.TARGET.SCALED

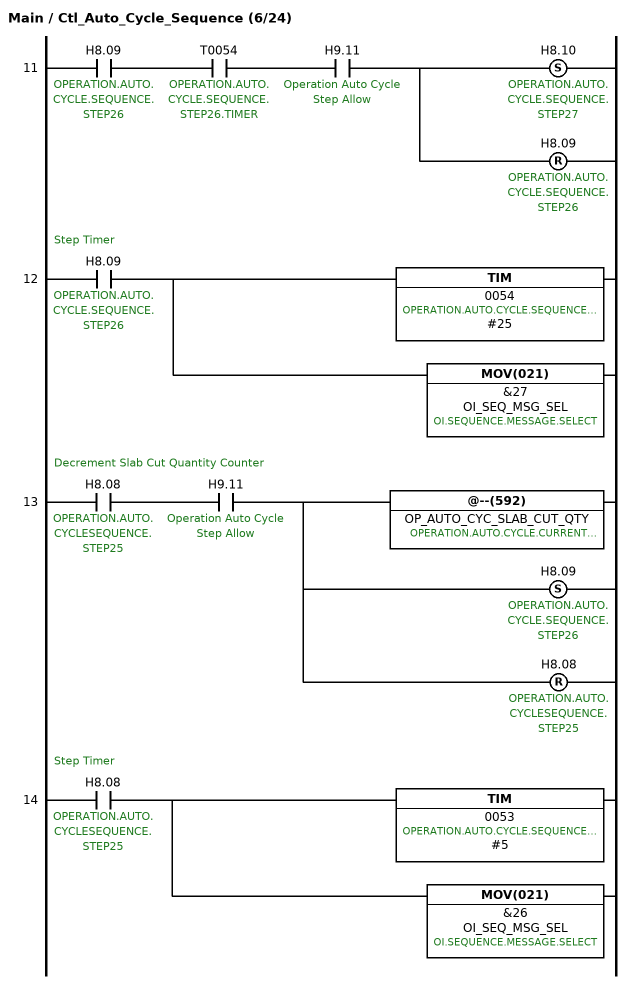
; rung 11
LD H8.09  ; OPERATION.AUTO.CYCLE.SEQUENCE.STEP26
AND T0054  ; OPERATION.AUTO.CYCLE.SEQUENCE.STEP26.TIMER
AND H9.11  ; Operation Auto Cycle Step Allow
SET H8.10  ; OPERATION.AUTO.CYCLE.SEQUENCE.STEP27
RSET H8.09  ; OPERATION.AUTO.CYCLE.SEQUENCE.STEP26
; rung 12: Step Timer
LD H8.09  ; OPERATION.AUTO.CYCLE.SEQUENCE.STEP26
TIM 0054 #25  ; OPERATION.AUTO.CYCLE.SEQUENCE.STEP26.TIMER
MOV(021) &27 OI_SEQ_MSG_SEL  ; OI.SEQUENCE.MESSAGE.SELECT
; rung 13: Decrement Slab Cut Quantity Counter
LD H8.08  ; OPERATION.AUTO.CYCLESEQUENCE.STEP25
AND H9.11  ; Operation Auto Cycle Step Allow
@--(592) OP_AUTO_CYC_SLAB_CUT_QTY  ; OPERATION.AUTO.CYCLE.CURRENT.SLAB.CUT.QUANTITY
SET H8.09  ; OPERATION.AUTO.CYCLE.SEQUENCE.STEP26
RSET H8.08  ; OPERATION.AUTO.CYCLESEQUENCE.STEP25
; rung 14: Step Timer
LD H8.08  ; OPERATION.AUTO.CYCLESEQUENCE.STEP25
TIM 0053 #5  ; OPERATION.AUTO.CYCLE.SEQUENCE.STEP25.TIMER
MOV(021) &26 OI_SEQ_MSG_SEL  ; OI.SEQUENCE.MESSAGE.SELECT

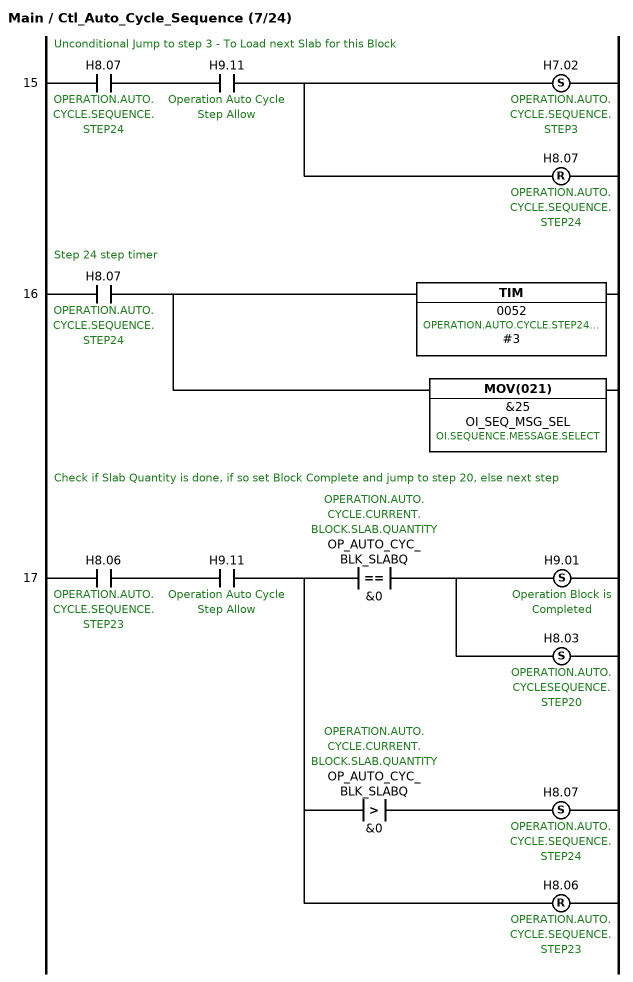
; rung 15: Unconditional Jump to step 3 - To Load next Slab for this Block
LD H8.07  ; OPERATION.AUTO.CYCLE.SEQUENCE.STEP24
AND H9.11  ; Operation Auto Cycle Step Allow
SET H7.02  ; OPERATION.AUTO.CYCLE.SEQUENCE.STEP3
RSET H8.07  ; OPERATION.AUTO.CYCLE.SEQUENCE.STEP24
; rung 16: Step 24 step timer
LD H8.07  ; OPERATION.AUTO.CYCLE.SEQUENCE.STEP24
TIM 0052 #3  ; OPERATION.AUTO.CYCLE.STEP24.TIMER
MOV(021) &25 OI_SEQ_MSG_SEL  ; OI.SEQUENCE.MESSAGE.SELECT
; rung 17: Check if Slab Quantity is done, if so set Block Complete and jump to step 20, else next step
LD H8.06  ; OPERATION.AUTO.CYCLE.SEQUENCE.STEP23
AND H9.11  ; Operation Auto Cycle Step Allow
OUT TR0
AND=(300) OP_AUTO_CYC_BLK_SLABQ &0  ; OPERATION.AUTO.CYCLE.CURRENT.BLOCK.SLAB.QUANTITY
SET H9.01  ; Operation Block is Completed
SET H8.03  ; OPERATION.AUTO.CYCLESEQUENCE.STEP20
LD TR0
AND>(320) OP_AUTO_CYC_BLK_SLABQ &0  ; OPERATION.AUTO.CYCLE.CURRENT.BLOCK.SLAB.QUANTITY
SET H8.07  ; OPERATION.AUTO.CYCLE.SEQUENCE.STEP24
LD TR0
RSET H8.06  ; OPERATION.AUTO.CYCLE.SEQUENCE.STEP23

